LIN {X 0,Y 530.391,Z 772.549,A -85,B 0,C 180,E1 -4220.081,E2 -4220.081} C_VEL
LIN {X 0,Y 530.37,Z 771.261,A -85,B 0,C 180,E1 -4220.851,E2 -4220.851} C_VEL
LIN {X 0,Y 530.472,Z 768.514,A -85,B 0,C 180,E1 -4222.004,E2 -4222.004} C_VEL
LIN {X 0,Y 530.565,Z 764.749,A -85,B 0,C 180,E1 -4223.153,E2 -4223.153} C_VEL
LIN {X 0,Y 530.601,Z 759.88,A -85,B 0,C 180,E1 -4224.299,E2 -4224.299} C_VEL
LIN {X 0,Y 530.713,Z 753.762,A -85,B 0,C 180,E1 -4225.443,E2 -4225.443} C_VEL
LIN {X 0,Y 530.767,Z 746.143,A -85,B 0,C 180,E1 -4226.584,E2 -4226.584} C_VEL
LIN {X 0,Y 531.037,Z 736.67,A -85,B 0,C 180,E1 -4227.725,E2 -4227.725} C_VEL
LIN {X 0,Y 531.27,Z 726.885,A -85,B 0,C 180,E1 -4228.674,E2 -4228.674} C_VEL
LIN {X 0,Y 531.461,Z 715.977,A -85,B 0,C 180,E1 -4229.526,E2 -4229.526} C_VEL
LIN {X 0,Y 531.816,Z 705.381,A -85,B 0,C 180,E1 -4230.189,E2 -4230.189} C_VEL
LIN {X 0,Y 532.07,Z 693.777,A -85,B 0,C 180,E1 -4230.757,E2 -4230.757} C_VEL
LIN {X 0,Y 532.235,Z 680.391,A -85,B 0,C 180,E1 -4231.229,E2 -4231.229} C_VEL
LIN {X 0,Y 532.411,Z 668.005,A -85,B 0,C 180,E1 -4231.513,E2 -4231.513} C_VEL
LIN {X 0,Y 532.675,Z 572.814,A -85,B 0,C 180,E1 -4232.812,E2 -4232.812} C_VEL
LIN {X 0,Y 531.118,Z 564.327,A -85,B 0,C 180,E1 -4232.987,E2 -4232.987} C_VEL
LIN {X 0,Y 531.078,Z 564.336,A -85,B 0,C 180,E1 -4236.077,E2 -4236.077} C_VEL
LIN {X 0,Y 531.019,Z 564.334,A -85,B 0,C 180,E1 -4239.138,E2 -4239.138} C_VEL
LIN {X 0,Y 531.044,Z 564.337,A -85,B 0,C 180,E1 -4242.225,E2 -4242.225} C_VEL
LIN {X 0,Y 530.998,Z 564.337,A -85,B 0,C 180,E1 -4245.349,E2 -4245.349} C_VEL
LIN {X 0,Y 530.991,Z 564.34,A -85,B 0,C 180,E1 -4248.521,E2 -4248.521} C_VEL
LIN {X 0,Y 531.001,Z 564.335,A -85,B 0,C 180,E1 -4250.937,E2 -4250.937} C_VEL
LIN {X 0,Y 530.966,Z 564.347,A -85,B 0,C 180,E1 -4254.225,E2 -4254.225} C_VEL
LIN {X 0,Y 531.006,Z 564.337,A -85,B 0,C 180,E1 -4256.743,E2 -4256.743} C_VEL
LIN {X 0,Y 530.99,Z 564.341,A -85,B 0,C 180,E1 -4259.321,E2 -4259.321} C_VEL
LIN {X 0,Y 531.056,Z 564.335,A -85,B 0,C 180,E1 -4261.1,E2 -4261.1} C_VEL
LIN {X 0,Y 532.797,Z 573.387,A -85,B 0,C 180,E1 -4261.29,E2 -4261.29} C_VEL
LIN {X 0,Y 532.448,Z 668.31,A -85,B 0,C 180,E1 -4262.594,E2 -4262.594} C_VEL
LIN {X 0,Y 532.309,Z 677.915,A -85,B 0,C 180,E1 -4262.8,E2 -4262.8} C_VEL
LIN {X 0,Y 532.099,Z 688.32,A -85,B 0,C 180,E1 -4263.125,E2 -4263.125} C_VEL
LIN {X 0,Y 531.952,Z 697.951,A -85,B 0,C 180,E1 -4263.527,E2 -4263.527} C_VEL
LIN {X 0,Y 531.753,Z 707.979,A -85,B 0,C 180,E1 -4264.059,E2 -4264.059} C_VEL
LIN {X 0,Y 531.543,Z 717.033,A -85,B 0,C 180,E1 -4264.648,E2 -4264.648} C_VEL
LIN {X 0,Y 531.302,Z 725.688,A -85,B 0,C 180,E1 -4265.322,E2 -4265.322} C_VEL
LIN {X 0,Y 531.151,Z 733.257,A -85,B 0,C 180,E1 -4266.019,E2 -4266.019} C_VEL
LIN {X 0,Y 530.967,Z 740.423,A -85,B 0,C 180,E1 -4266.793,E2 -4266.793} C_VEL
LIN {X 0,Y 530.801,Z 747.91,A -85,B 0,C 180,E1 -4267.76,E2 -4267.76} C_VEL
LIN {X 0,Y 530.68,Z 754.502,A -85,B 0,C 180,E1 -4268.788,E2 -4268.788} C_VEL
LIN {X 0,Y 530.604,Z 759.873,A -85,B 0,C 180,E1 -4269.805,E2 -4269.805} C_VEL
LIN {X 0,Y 530.529,Z 762.94,A -85,B 0,C 180,E1 -4270.473,E2 -4270.473} C_VEL
LIN {X 0,Y 530.489,Z 766.691,A -85,B 0,C 180,E1 -4271.482,E2 -4271.482} C_VEL
LIN {X 0,Y 530.427,Z 769.651,A -85,B 0,C 180,E1 -4272.51,E2 -4272.51} C_VEL
LIN {X 0,Y 530.357,Z 771.836,A -85,B 0,C 180,E1 -4273.556,E2 -4273.556} C_VEL
LIN {X 0,Y 530.379,Z 773.243,A -85,B 0,C 180,E1 -4274.61,E2 -4274.61} C_VEL
LIN {X 0,Y 530.38,Z 773.892,A -85,B 0,C 180,E1 -4275.687,E2 -4275.687} C_VEL
LIN {X 0,Y 530.334,Z 773.739,A -85,B 0,C 180,E1 -4276.789,E2 -4276.789} C_VEL
LIN {X 0,Y 530.388,Z 772.739,A -85,B 0,C 180,E1 -4277.904,E2 -4277.904} C_VEL
LIN {X 0,Y 530.375,Z 770.803,A -85,B 0,C 180,E1 -4279.051,E2 -4279.051} C_VEL
LIN {X 0,Y 530.43,Z 767.85,A -85,B 0,C 180,E1 -4280.216,E2 -4280.216} C_VEL
LIN {X 0,Y 530.517,Z 762.445,A -85,B 0,C 180,E1 -4281.733,E2 -4281.733} C_VEL
LIN {X 0,Y 530.587,Z 757.227,A -85,B 0,C 180,E1 -4282.824,E2 -4282.824} C_VEL
LIN {X 0,Y 530.726,Z 751.007,A -85,B 0,C 180,E1 -4283.877,E2 -4283.877} C_VEL
LIN {X 0,Y 530.847,Z 744.546,A -85,B 0,C 180,E1 -4284.79,E2 -4284.79} C_VEL
LIN {X 0,Y 531.056,Z 737.211,A -85,B 0,C 180,E1 -4285.66,E2 -4285.66} C_VEL
LIN {X 0,Y 531.242,Z 728.486,A -85,B 0,C 180,E1 -4286.523,E2 -4286.523} C_VEL
LIN {X 0,Y 531.461,Z 719.636,A -85,B 0,C 180,E1 -4287.252,E2 -4287.252} C_VEL
LIN {X 0,Y 531.674,Z 710.874,A -85,B 0,C 180,E1 -4287.856,E2 -4287.856} C_VEL
LIN {X 0,Y 531.865,Z 701.897,A -85,B 0,C 180,E1 -4288.37,E2 -4288.37} C_VEL
LIN {X 0,Y 532.04,Z 691.985,A -85,B 0,C 180,E1 -4288.825,E2 -4288.825} C_VEL
LIN {X 0,Y 532.229,Z 681.54,A -85,B 0,C 180,E1 -4289.19,E2 -4289.19} C_VEL
LIN {X 0,Y 532.326,Z 671.036,A -85,B 0,C 180,E1 -4289.45,E2 -4289.45} C_VEL
LIN {X 0,Y 532.497,Z 646.041,A -85,B 0,C 180,E1 -4289.817,E2 -4289.817} C_VEL
LIN {X 0,Y 532.659,Z 574.015,A -85,B 0,C 180,E1 -4290.795,E2 -4290.795} C_VEL
LIN {X 0,Y 531.05,Z 565.236,A -85,B 0,C 180,E1 -4290.985,E2 -4290.985} C_VEL
LIN {X 0,Y 530.982,Z 564.345,A -85,B 0,C 180,E1 -4291.244,E2 -4291.244} C_VEL
LIN {X 0,Y 531.008,Z 564.342,A -85,B 0,C 180,E1 -4294.154,E2 -4294.154} C_VEL
LIN {X 0,Y 530.957,Z 564.35,A -85,B 0,C 180,E1 -4296.603,E2 -4296.603} C_VEL
LIN {X 0,Y 531.015,Z 564.337,A -85,B 0,C 180,E1 -4299.872,E2 -4299.872} C_VEL
LIN {X 0,Y 530.983,Z 564.341,A -85,B 0,C 180,E1 -4303.071,E2 -4303.071} C_VEL
LIN {X 0,Y 531.009,Z 564.336,A -85,B 0,C 180,E1 -4305.436,E2 -4305.436} C_VEL
LIN {X 0,Y 531.037,Z 564.34,A -85,B 0,C 180,E1 -4308.55,E2 -4308.55} C_VEL
LIN {X 0,Y 531.052,Z 564.33,A -85,B 0,C 180,E1 -4311.629,E2 -4311.629} C_VEL
LIN {X 0,Y 531.132,Z 564.327,A -85,B 0,C 180,E1 -4314.685,E2 -4314.685} C_VEL
LIN {X 0,Y 531.13,Z 564.32,A -85,B 0,C 180,E1 -4317.725,E2 -4317.725} C_VEL
LIN {X 0,Y 531.146,Z 564.324,A -85,B 0,C 180,E1 -4320.758,E2 -4320.758} C_VEL
LIN {X 0,Y 531.1,Z 564.325,A -85,B 0,C 180,E1 -4323.034,E2 -4323.034} C_VEL
LIN {X 0,Y 531.081,Z 564.329,A -85,B 0,C 180,E1 -4326.077,E2 -4326.077} C_VEL
LIN {X 0,Y 531.027,Z 564.333,A -85,B 0,C 180,E1 -4329.138,E2 -4329.138} C_VEL
LIN {X 0,Y 531.031,Z 564.336,A -85,B 0,C 180,E1 -4332.225,E2 -4332.225} C_VEL
LIN {X 0,Y 530.986,Z 564.337,A -85,B 0,C 180,E1 -4335.35,E2 -4335.35} C_VEL
LIN {X 0,Y 531.007,Z 564.333,A -85,B 0,C 180,E1 -4337.723,E2 -4337.723} C_VEL
LIN {X 0,Y 530.996,Z 564.339,A -85,B 0,C 180,E1 -4340.938,E2 -4340.938} C_VEL
LIN {X 0,Y 530.999,Z 564.338,A -85,B 0,C 180,E1 -4344.046,E2 -4344.046} C_VEL
LIN {X 0,Y 531.004,Z 564.34,A -85,B 0,C 180,E1 -4346.744,E2 -4346.744} C_VEL
LIN {X 0,Y 530.993,Z 564.338,A -85,B 0,C 180,E1 -4349.322,E2 -4349.322} C_VEL
LIN {X 0,Y 530.973,Z 564.343,A -85,B 0,C 180,E1 -4352.104,E2 -4352.104} C_VEL
LIN {X 0,Y 530.984,Z 564.343,A -85,B 0,C 180,E1 -4354.855,E2 -4354.855} C_VEL
LIN {X 0,Y 530.962,Z 564.341,A -85,B 0,C 180,E1 -4357.508,E2 -4357.508} C_VEL
LIN {X 0,Y 531.021,Z 564.342,A -85,B 0,C 180,E1 -4360.429,E2 -4360.429} C_VEL
LIN {X 0,Y 530.963,Z 564.341,A -85,B 0,C 180,E1 -4363.495,E2 -4363.495} C_VEL
LIN {X 0,Y 530.955,Z 564.351,A -85,B 0,C 180,E1 -4366.506,E2 -4366.506} C_VEL
LIN {X 0,Y 530.986,Z 564.341,A -85,B 0,C 180,E1 -4368.977,E2 -4368.977} C_VEL
LIN {X 0,Y 530.957,Z 564.342,A -85,B 0,C 180,E1 -4371.53,E2 -4371.53} C_VEL
LIN {X 0,Y 530.961,Z 564.35,A -85,B 0,C 180,E1 -4374.381,E2 -4374.381} C_VEL
LIN {X 0,Y 530.969,Z 564.343,A -85,B 0,C 180,E1 -4377.134,E2 -4377.134} C_VEL
LIN {X 0,Y 530.968,Z 564.343,A -85,B 0,C 180,E1 -4379.804,E2 -4379.804} C_VEL
LIN {X 0,Y 531.015,Z 564.344,A -85,B 0,C 180,E1 -4382.468,E2 -4382.468} C_VEL
LIN {X 0,Y 531.004,Z 564.377,A -85,B 0,C 180,E1 -4383.519,E2 -4383.519} C_VEL
LIN {X 0,Y 532.974,Z 574.901,A -85,B 0,C 180,E1 -4385.042,E2 -4385.042} C_VEL
LIN {X 0,Y 532.626,Z 593.287,A -85,B 0,C 180,E1 -4387.502,E2 -4387.502} C_VEL
LIN {X 0,Y 532.157,Z 617.709,A -85,B 0,C 180,E1 -4390.722,E2 -4390.722} C_VEL
LIN {X 0,Y 531.683,Z 641.975,A -85,B 0,C 180,E1 -4393.884,E2 -4393.884} C_VEL
LIN {X 0,Y 531.55,Z 650.859,A -85,B 0,C 180,E1 -4395.042,E2 -4395.042} C_VEL
LIN {X 0,Y 532.848,Z 660.029,A -85,B 0,C 180,E1 -4395.204,E2 -4395.204} C_VEL
LIN {X 0,Y 532.474,Z 759.96,A -85,B 0,C 180,E1 -4396.573,E2 -4396.573} C_VEL
LIN {X 0,Y 532.254,Z 772.456,A -85,B 0,C 180,E1 -4396.883,E2 -4396.883} C_VEL
LIN {X 0,Y 532.024,Z 785.368,A -85,B 0,C 180,E1 -4397.362,E2 -4397.362} C_VEL
LIN {X 0,Y 531.807,Z 797.309,A -85,B 0,C 180,E1 -4397.967,E2 -4397.967} C_VEL
LIN {X 0,Y 531.526,Z 809.198,A -85,B 0,C 180,E1 -4398.754,E2 -4398.754} C_VEL
LIN {X 0,Y 531.255,Z 819.607,A -85,B 0,C 180,E1 -4399.616,E2 -4399.616} C_VEL
LIN {X 0,Y 531.06,Z 828.116,A -85,B 0,C 180,E1 -4400.478,E2 -4400.478} C_VEL
LIN {X 0,Y 530.886,Z 835.962,A -85,B 0,C 180,E1 -4401.435,E2 -4401.435} C_VEL
LIN {X 0,Y 530.685,Z 843.623,A -85,B 0,C 180,E1 -4402.581,E2 -4402.581} C_VEL
LIN {X 0,Y 530.604,Z 850.679,A -85,B 0,C 180,E1 -4403.918,E2 -4403.918} C_VEL
LIN {X 0,Y 530.459,Z 855.372,A -85,B 0,C 180,E1 -4405.06,E2 -4405.06} C_VEL
LIN {X 0,Y 530.516,Z 858.961,A -85,B 0,C 180,E1 -4406.202,E2 -4406.202} C_VEL
LIN {X 0,Y 530.457,Z 860.81,A -85,B 0,C 180,E1 -4406.962,E2 -4406.962} C_VEL
LIN {X 0,Y 530.41,Z 862.197,A -85,B 0,C 180,E1 -4407.722,E2 -4407.722} C_VEL
LIN {X 0,Y 530.344,Z 863.786,A -85,B 0,C 180,E1 -4409.241,E2 -4409.241} C_VEL
LIN {X 0,Y 530.342,Z 864,A -85,B 0,C 180,E1 -4410,E2 -4410} C_VEL
LIN {X 0,Y 530.361,Z 863.183,A -85,B 0,C 180,E1 -4411.519,E2 -4411.519} C_VEL
LIN {X 0,Y 530.41,Z 862.194,A -85,B 0,C 180,E1 -4412.278,E2 -4412.278} C_VEL
LIN {X 0,Y 530.457,Z 860.807,A -85,B 0,C 180,E1 -4413.038,E2 -4413.038} C_VEL
LIN {X 0,Y 530.523,Z 857.895,A -85,B 0,C 180,E1 -4414.178,E2 -4414.178} C_VEL
LIN {X 0,Y 530.525,Z 853.95,A -85,B 0,C 180,E1 -4415.321,E2 -4415.321} C_VEL
LIN {X 0,Y 530.599,Z 848.264,A -85,B 0,C 180,E1 -4416.582,E2 -4416.582} C_VEL
LIN {X 0,Y 530.758,Z 841.237,A -85,B 0,C 180,E1 -4417.8,E2 -4417.8} C_VEL
LIN {X 0,Y 530.93,Z 832.994,A -85,B 0,C 180,E1 -4418.948,E2 -4418.948} C_VEL
LIN {X 0,Y 531.137,Z 824.542,A -85,B 0,C 180,E1 -4419.905,E2 -4419.905} C_VEL
LIN {X 0,Y 531.408,Z 814.096,A -85,B 0,C 180,E1 -4420.863,E2 -4420.863} C_VEL
LIN {X 0,Y 531.667,Z 802.16,A -85,B 0,C 180,E1 -4421.737,E2 -4421.737} C_VEL
LIN {X 0,Y 531.95,Z 790.496,A -85,B 0,C 180,E1 -4422.397,E2 -4422.397} C_VEL
LIN {X 0,Y 532.205,Z 778.182,A -85,B 0,C 180,E1 -4422.924,E2 -4422.924} C_VEL
LIN {X 0,Y 532.353,Z 765.533,A -85,B 0,C 180,E1 -4423.309,E2 -4423.309} C_VEL
LIN {X 0,Y 532.491,Z 752.335,A -85,B 0,C 180,E1 -4423.548,E2 -4423.548} C_VEL
LIN {X 0,Y 532.701,Z 656.891,A -85,B 0,C 180,E1 -4424.843,E2 -4424.843} C_VEL
LIN {X 0,Y 531.719,Z 649.794,A -85,B 0,C 180,E1 -4424.977,E2 -4424.977} C_VEL
LIN {X 0,Y 532.246,Z 621.608,A -85,B 0,C 180,E1 -4428.199,E2 -4428.199} C_VEL
LIN {X 0,Y 532.815,Z 595.021,A -85,B 0,C 180,E1 -4431.268,E2 -4431.268} C_VEL
LIN {X 0,Y 533.193,Z 575.94,A -85,B 0,C 180,E1 -4433.498,E2 -4433.498} C_VEL
LIN {X 0,Y 532.837,Z 572.446,A -85,B 0,C 180,E1 -4433.927,E2 -4433.927} C_VEL
LIN {X 0,Y 531.05,Z 564.336,A -85,B 0,C 180,E1 -4435.002,E2 -4435.002} C_VEL
LIN {X 0,Y 531.018,Z 564.34,A -85,B 0,C 180,E1 -4437.595,E2 -4437.595} C_VEL
LIN {X 0,Y 530.973,Z 564.341,A -85,B 0,C 180,E1 -4440.644,E2 -4440.644} C_VEL
LIN {X 0,Y 530.992,Z 564.344,A -85,B 0,C 180,E1 -4443.771,E2 -4443.771} C_VEL
LIN {X 0,Y 530.966,Z 564.343,A -85,B 0,C 180,E1 -4446.557,E2 -4446.557} C_VEL
LIN {X 0,Y 531.004,Z 564.341,A -85,B 0,C 180,E1 -4449.857,E2 -4449.857} C_VEL
LIN {X 0,Y 530.977,Z 564.343,A -85,B 0,C 180,E1 -4452.456,E2 -4452.456} C_VEL
LIN {X 0,Y 530.983,Z 564.339,A -85,B 0,C 180,E1 -4455.62,E2 -4455.62} C_VEL
LIN {X 0,Y 531.004,Z 564.338,A -85,B 0,C 180,E1 -4458.565,E2 -4458.565} C_VEL
LIN {X 0,Y 530.964,Z 564.339,A -85,B 0,C 180,E1 -4461.345,E2 -4461.345} C_VEL
LIN {X 0,Y 530.976,Z 564.343,A -85,B 0,C 180,E1 -4464.381,E2 -4464.381} C_VEL
LIN {X 0,Y 530.965,Z 564.34,A -85,B 0,C 180,E1 -4467.133,E2 -4467.133} C_VEL
LIN {X 0,Y 530.978,Z 564.34,A -85,B 0,C 180,E1 -4469.803,E2 -4469.803} C_VEL
LIN {X 0,Y 531.01,Z 564.343,A -85,B 0,C 180,E1 -4472.466,E2 -4472.466} C_VEL
LIN {X 0,Y 530.999,Z 564.337,A -85,B 0,C 180,E1 -4474.942,E2 -4474.942} C_VEL
LIN {X 0,Y 530.962,Z 564.342,A -85,B 0,C 180,E1 -4478.246,E2 -4478.246} C_VEL
LIN {X 0,Y 530.988,Z 564.343,A -85,B 0,C 180,E1 -4480.677,E2 -4480.677} C_VEL
LIN {X 0,Y 530.982,Z 564.336,A -85,B 0,C 180,E1 -4483.071,E2 -4483.071} C_VEL
LIN {X 0,Y 531.009,Z 564.333,A -85,B 0,C 180,E1 -4485.436,E2 -4485.436} C_VEL
LIN {X 0,Y 531.037,Z 564.34,A -85,B 0,C 180,E1 -4488.55,E2 -4488.55} C_VEL
LIN {X 0,Y 531.05,Z 564.325,A -85,B 0,C 180,E1 -4491.629,E2 -4491.629} C_VEL
LIN {X 0,Y 531.136,Z 564.328,A -85,B 0,C 180,E1 -4494.685,E2 -4494.685} C_VEL
LIN {X 0,Y 531.13,Z 564.315,A -85,B 0,C 180,E1 -4497.725,E2 -4497.725} C_VEL
LIN {X 0,Y 531.148,Z 564.326,A -85,B 0,C 180,E1 -4500.758,E2 -4500.758} C_VEL
LIN {X 0,Y 531.1,Z 564.327,A -85,B 0,C 180,E1 -4503.034,E2 -4503.034} C_VEL
LIN {X 0,Y 531.081,Z 564.321,A -85,B 0,C 180,E1 -4506.077,E2 -4506.077} C_VEL
LIN {X 0,Y 531.027,Z 564.337,A -85,B 0,C 180,E1 -4509.138,E2 -4509.138} C_VEL
LIN {X 0,Y 531.031,Z 564.33,A -85,B 0,C 180,E1 -4512.225,E2 -4512.225} C_VEL
LIN {X 0,Y 530.986,Z 564.341,A -85,B 0,C 180,E1 -4515.35,E2 -4515.35} C_VEL
LIN {X 0,Y 531.007,Z 564.333,A -85,B 0,C 180,E1 -4517.723,E2 -4517.723} C_VEL
LIN {X 0,Y 530.993,Z 564.344,A -85,B 0,C 180,E1 -4520.938,E2 -4520.938} C_VEL
LIN {X 0,Y 530.971,Z 564.337,A -85,B 0,C 180,E1 -4524.225,E2 -4524.225} C_VEL
LIN {X 0,Y 531.004,Z 564.339,A -85,B 0,C 180,E1 -4526.744,E2 -4526.744} C_VEL
LIN {X 0,Y 530.992,Z 564.34,A -85,B 0,C 180,E1 -4529.322,E2 -4529.322} C_VEL
LIN {X 0,Y 530.972,Z 564.34,A -85,B 0,C 180,E1 -4532.104,E2 -4532.104} C_VEL
LIN {X 0,Y 530.981,Z 564.341,A -85,B 0,C 180,E1 -4534.855,E2 -4534.855} C_VEL
LIN {X 0,Y 530.967,Z 564.345,A -85,B 0,C 180,E1 -4537.508,E2 -4537.508} C_VEL
LIN {X 0,Y 530.979,Z 564.338,A -85,B 0,C 180,E1 -4540.433,E2 -4540.433} C_VEL
LIN {X 0,Y 530.966,Z 564.343,A -85,B 0,C 180,E1 -4543.283,E2 -4543.283} C_VEL
LIN {X 0,Y 530.959,Z 564.346,A -85,B 0,C 180,E1 -4543.581,E2 -4543.581} C_VEL
LIN {X 0,Y 530.285,Z 564.427,A -85,B 0,C 180,E1 -4544.214,E2 -4544.214} C_VEL
LIN {X 0,Y 527.432,Z 564.789,A -85,B 0,C 180,E1 -4545.243,E2 -4545.243} C_VEL
LIN {X 0,Y 525.026,Z 565.087,A -85,B 0,C 180,E1 -4546.071,E2 -4546.071} C_VEL
LIN {X 0,Y 523.994,Z 565.211,A -85,B 0,C 180,E1 -4546.711,E2 -4546.711} C_VEL
LIN {X 0,Y 523.91,Z 565.22,A -85,B 0,C 180,E1 -4546.928,E2 -4546.928} C_VEL
LIN {X 0,Y 523.945,Z 565.218,A -85,B 0,C 180,E1 -4549.921,E2 -4549.921} C_VEL
LIN {X 0,Y 523.909,Z 565.219,A -85,B 0,C 180,E1 -4552.869,E2 -4552.869} C_VEL
LIN {X 0,Y 523.942,Z 565.221,A -85,B 0,C 180,E1 -4555.711,E2 -4555.711} C_VEL
LIN {X 0,Y 523.922,Z 565.218,A -85,B 0,C 180,E1 -4558.457,E2 -4558.457} C_VEL
LIN {X 0,Y 523.939,Z 565.221,A -85,B 0,C 180,E1 -4561.126,E2 -4561.126} C_VEL
LIN {X 0,Y 523.961,Z 565.371,A -85,B 0,C 180,E1 -4562.868,E2 -4562.868} C_VEL
LIN {X 0,Y 523.989,Z 565.59,A -85,B 0,C 180,E1 -4562.918,E2 -4562.918} C_VEL
LIN {X 0,Y 525.93,Z 575.467,A -85,B 0,C 180,E1 -4563.114,E2 -4563.114} C_VEL
LIN {X 0,Y 525.487,Z 671.22,A -85,B 0,C 180,E1 -4564.449,E2 -4564.449} C_VEL
LIN {X 0,Y 525.28,Z 683.407,A -85,B 0,C 180,E1 -4564.757,E2 -4564.757} C_VEL
LIN {X 0,Y 525.143,Z 695.77,A -85,B 0,C 180,E1 -4565.226,E2 -4565.226} C_VEL
LIN {X 0,Y 524.907,Z 707.21,A -85,B 0,C 180,E1 -4565.812,E2 -4565.812} C_VEL
LIN {X 0,Y 524.603,Z 717.948,A -85,B 0,C 180,E1 -4566.513,E2 -4566.513} C_VEL
LIN {X 0,Y 524.309,Z 727.575,A -85,B 0,C 180,E1 -4567.291,E2 -4567.291} C_VEL
LIN {X 0,Y 524.093,Z 736.326,A -85,B 0,C 180,E1 -4568.154,E2 -4568.154} C_VEL
LIN {X 0,Y 523.853,Z 744.814,A -85,B 0,C 180,E1 -4569.175,E2 -4569.175} C_VEL
LIN {X 0,Y 523.661,Z 753.01,A -85,B 0,C 180,E1 -4570.396,E2 -4570.396} C_VEL
LIN {X 0,Y 523.533,Z 759.515,A -85,B 0,C 180,E1 -4571.611,E2 -4571.611} C_VEL
LIN {X 0,Y 523.445,Z 764.578,A -85,B 0,C 180,E1 -4572.82,E2 -4572.82} C_VEL
LIN {X 0,Y 523.355,Z 768.482,A -85,B 0,C 180,E1 -4574.021,E2 -4574.021} C_VEL
LIN {X 0,Y 523.339,Z 771.289,A -85,B 0,C 180,E1 -4575.218,E2 -4575.218} C_VEL
LIN {X 0,Y 523.3,Z 772.591,A -85,B 0,C 180,E1 -4576.011,E2 -4576.011} C_VEL
LIN {X 0,Y 523.268,Z 773.482,A -85,B 0,C 180,E1 -4576.802,E2 -4576.802} C_VEL
LIN {X 0,Y 523.282,Z 773.913,A -85,B 0,C 180,E1 -4577.591,E2 -4577.591} C_VEL
LIN {X 0,Y 523.363,Z 773.892,A -85,B 0,C 180,E1 -4578.604,E2 -4578.604} C_VEL
LIN {X 0,Y 523.31,Z 772.783,A -85,B 0,C 180,E1 -4579.946,E2 -4579.946} C_VEL
LIN {X 0,Y 523.316,Z 769.939,A -85,B 0,C 180,E1 -4581.505,E2 -4581.505} C_VEL
LIN {X 0,Y 523.451,Z 766.663,A -85,B 0,C 180,E1 -4582.672,E2 -4582.672} C_VEL
LIN {X 0,Y 523.434,Z 762.367,A -85,B 0,C 180,E1 -4583.834,E2 -4583.834} C_VEL
LIN {X 0,Y 523.543,Z 755.905,A -85,B 0,C 180,E1 -4585.187,E2 -4585.187} C_VEL
LIN {X 0,Y 523.722,Z 748.867,A -85,B 0,C 180,E1 -4586.345,E2 -4586.345} C_VEL
LIN {X 0,Y 523.954,Z 740.148,A -85,B 0,C 180,E1 -4587.502,E2 -4587.502} C_VEL
LIN {X 0,Y 524.225,Z 730.125,A -85,B 0,C 180,E1 -4588.56,E2 -4588.56} C_VEL
LIN {X 0,Y 524.451,Z 720.028,A -85,B 0,C 180,E1 -4589.424,E2 -4589.424} C_VEL
LIN {X 0,Y 524.8,Z 708.697,A -85,B 0,C 180,E1 -4590.192,E2 -4590.192} C_VEL
LIN {X 0,Y 525.165,Z 695.762,A -85,B 0,C 180,E1 -4590.863,E2 -4590.863} C_VEL
LIN {X 0,Y 525.351,Z 683.831,A -85,B 0,C 180,E1 -4591.317,E2 -4591.317} C_VEL
LIN {X 0,Y 525.548,Z 670.515,A -85,B 0,C 180,E1 -4591.652,E2 -4591.652} C_VEL
LIN {X 0,Y 525.827,Z 573.57,A -85,B 0,C 180,E1 -4593.005,E2 -4593.005} C_VEL
LIN {X 0,Y 524.47,Z 566.934,A -85,B 0,C 180,E1 -4593.138,E2 -4593.138} C_VEL
LIN {X 0,Y 524.03,Z 565.211,A -85,B 0,C 180,E1 -4593.195,E2 -4593.195} C_VEL
LIN {X 0,Y 524.04,Z 565.212,A -85,B 0,C 180,E1 -4596.159,E2 -4596.159} C_VEL
LIN {X 0,Y 523.989,Z 565.211,A -85,B 0,C 180,E1 -4599.262,E2 -4599.262} C_VEL
LIN {X 0,Y 524.028,Z 565.209,A -85,B 0,C 180,E1 -4601.751,E2 -4601.751} C_VEL
LIN {X 0,Y 523.996,Z 565.209,A -85,B 0,C 180,E1 -4605.052,E2 -4605.052} C_VEL
LIN {X 0,Y 523.966,Z 565.221,A -85,B 0,C 180,E1 -4607.968,E2 -4607.968} C_VEL
LIN {X 0,Y 523.974,Z 565.215,A -85,B 0,C 180,E1 -4610.409,E2 -4610.409} C_VEL
LIN {X 0,Y 523.912,Z 565.219,A -85,B 0,C 180,E1 -4612.893,E2 -4612.893} C_VEL
LIN {X 0,Y 523.985,Z 565.219,A -85,B 0,C 180,E1 -4616.019,E2 -4616.019} C_VEL
LIN {X 0,Y 523.942,Z 565.218,A -85,B 0,C 180,E1 -4618.874,E2 -4618.874} C_VEL
LIN {X 0,Y 524.023,Z 565.211,A -85,B 0,C 180,E1 -4620.911,E2 -4620.911} C_VEL
LIN {X 0,Y 525.834,Z 573.683,A -85,B 0,C 180,E1 -4621.09,E2 -4621.09} C_VEL
LIN {X 0,Y 525.495,Z 670.324,A -85,B 0,C 180,E1 -4622.443,E2 -4622.443} C_VEL
LIN {X 0,Y 525.388,Z 680.701,A -85,B 0,C 180,E1 -4622.69,E2 -4622.69} C_VEL
LIN {X 0,Y 525.224,Z 690.839,A -85,B 0,C 180,E1 -4623.034,E2 -4623.034} C_VEL
LIN {X 0,Y 524.988,Z 701.004,A -85,B 0,C 180,E1 -4623.487,E2 -4623.487} C_VEL
LIN {X 0,Y 524.796,Z 710.378,A -85,B 0,C 180,E1 -4624.015,E2 -4624.015} C_VEL
LIN {X 0,Y 524.566,Z 718.82,A -85,B 0,C 180,E1 -4624.591,E2 -4624.591} C_VEL
LIN {X 0,Y 524.342,Z 726.302,A -85,B 0,C 180,E1 -4625.193,E2 -4625.193} C_VEL
LIN {X 0,Y 524.149,Z 733.941,A -85,B 0,C 180,E1 -4625.916,E2 -4625.916} C_VEL
LIN {X 0,Y 523.95,Z 741.311,A -85,B 0,C 180,E1 -4626.741,E2 -4626.741} C_VEL
LIN {X 0,Y 523.755,Z 748.192,A -85,B 0,C 180,E1 -4627.656,E2 -4627.656} C_VEL
LIN {X 0,Y 523.622,Z 754.623,A -85,B 0,C 180,E1 -4628.687,E2 -4628.687} C_VEL
LIN {X 0,Y 523.545,Z 759.332,A -85,B 0,C 180,E1 -4629.588,E2 -4629.588} C_VEL
LIN {X 0,Y 523.436,Z 763.807,A -85,B 0,C 180,E1 -4630.63,E2 -4630.63} C_VEL
LIN {X 0,Y 523.389,Z 767.452,A -85,B 0,C 180,E1 -4631.678,E2 -4631.678} C_VEL
LIN {X 0,Y 523.333,Z 769.437,A -85,B 0,C 180,E1 -4632.386,E2 -4632.386} C_VEL
LIN {X 0,Y 523.258,Z 771.8,A -85,B 0,C 180,E1 -4633.507,E2 -4633.507} C_VEL
LIN {X 0,Y 523.279,Z 773.266,A -85,B 0,C 180,E1 -4634.616,E2 -4634.616} C_VEL
LIN {X 0,Y 523.279,Z 773.892,A -85,B 0,C 180,E1 -4635.701,E2 -4635.701} C_VEL
LIN {X 0,Y 523.239,Z 773.746,A -85,B 0,C 180,E1 -4636.763,E2 -4636.763} C_VEL
LIN {X 0,Y 523.309,Z 772.863,A -85,B 0,C 180,E1 -4637.817,E2 -4637.817} C_VEL
LIN {X 0,Y 523.305,Z 770.274,A -85,B 0,C 180,E1 -4639.356,E2 -4639.356} C_VEL
LIN {X 0,Y 523.402,Z 765.974,A -85,B 0,C 180,E1 -4640.869,E2 -4640.869} C_VEL
LIN {X 0,Y 523.471,Z 760.957,A -85,B 0,C 180,E1 -4642.146,E2 -4642.146} C_VEL
LIN {X 0,Y 523.553,Z 756.582,A -85,B 0,C 180,E1 -4643.052,E2 -4643.052} C_VEL
LIN {X 0,Y 523.706,Z 750.78,A -85,B 0,C 180,E1 -4644.047,E2 -4644.047} C_VEL
LIN {X 0,Y 523.874,Z 743.466,A -85,B 0,C 180,E1 -4645.081,E2 -4645.081} C_VEL
LIN {X 0,Y 524.104,Z 736.851,A -85,B 0,C 180,E1 -4645.867,E2 -4645.867} C_VEL
LIN {X 0,Y 524.292,Z 728.984,A -85,B 0,C 180,E1 -4646.661,E2 -4646.661} C_VEL
LIN {X 0,Y 524.525,Z 720.38,A -85,B 0,C 180,E1 -4647.387,E2 -4647.387} C_VEL
LIN {X 0,Y 524.766,Z 710.679,A -85,B 0,C 180,E1 -4648.061,E2 -4648.061} C_VEL
LIN {X 0,Y 524.967,Z 701.452,A -85,B 0,C 180,E1 -4648.585,E2 -4648.585} C_VEL
LIN {X 0,Y 525.158,Z 691.073,A -85,B 0,C 180,E1 -4649.052,E2 -4649.052} C_VEL
LIN {X 0,Y 525.334,Z 680.742,A -85,B 0,C 180,E1 -4649.402,E2 -4649.402} C_VEL
LIN {X 0,Y 525.471,Z 670.156,A -85,B 0,C 180,E1 -4649.652,E2 -4649.652} C_VEL
LIN {X 0,Y 525.874,Z 575.325,A -85,B 0,C 180,E1 -4650.976,E2 -4650.976} C_VEL
LIN {X 0,Y 524.083,Z 566.116,A -85,B 0,C 180,E1 -4651.161,E2 -4651.161} C_VEL
LIN {X 0,Y 523.96,Z 565.22,A -85,B 0,C 180,E1 -4651.4,E2 -4651.4} C_VEL
LIN {X 0,Y 523.977,Z 565.216,A -85,B 0,C 180,E1 -4653.979,E2 -4653.979} C_VEL
LIN {X 0,Y 523.928,Z 565.224,A -85,B 0,C 180,E1 -4656.27,E2 -4656.27} C_VEL
LIN {X 0,Y 523.938,Z 565.223,A -85,B 0,C 180,E1 -4658.766,E2 -4658.766} C_VEL
LIN {X 0,Y 523.945,Z 565.217,A -85,B 0,C 180,E1 -4661.22,E2 -4661.22} C_VEL
LIN {X 0,Y 523.931,Z 565.218,A -85,B 0,C 180,E1 -4663.639,E2 -4663.639} C_VEL
LIN {X 0,Y 523.932,Z 565.22,A -85,B 0,C 180,E1 -4666.028,E2 -4666.028} C_VEL
LIN {X 0,Y 524.001,Z 565.216,A -85,B 0,C 180,E1 -4668.394,E2 -4668.394} C_VEL
LIN {X 0,Y 523.999,Z 565.209,A -85,B 0,C 180,E1 -4671.516,E2 -4671.516} C_VEL
LIN {X 0,Y 524.09,Z 565.204,A -85,B 0,C 180,E1 -4674.614,E2 -4674.614} C_VEL
LIN {X 0,Y 524.102,Z 565.195,A -85,B 0,C 180,E1 -4677.694,E2 -4677.694} C_VEL
LIN {X 0,Y 524.115,Z 565.2,A -85,B 0,C 180,E1 -4680.768,E2 -4680.768} C_VEL
LIN {X 0,Y 524.067,Z 565.2,A -85,B 0,C 180,E1 -4683.075,E2 -4683.075} C_VEL
LIN {X 0,Y 524.042,Z 565.207,A -85,B 0,C 180,E1 -4686.159,E2 -4686.159} C_VEL
LIN {X 0,Y 523.995,Z 565.208,A -85,B 0,C 180,E1 -4689.262,E2 -4689.262} C_VEL
LIN {X 0,Y 524.014,Z 565.206,A -85,B 0,C 180,E1 -4691.752,E2 -4691.752} C_VEL
LIN {X 0,Y 523.983,Z 565.211,A -85,B 0,C 180,E1 -4695.053,E2 -4695.053} C_VEL
LIN {X 0,Y 523.955,Z 565.213,A -85,B 0,C 180,E1 -4697.969,E2 -4697.969} C_VEL
LIN {X 0,Y 523.964,Z 565.218,A -85,B 0,C 180,E1 -4700.41,E2 -4700.41} C_VEL
LIN {X 0,Y 523.935,Z 565.218,A -85,B 0,C 180,E1 -4702.893,E2 -4702.893} C_VEL
LIN {X 0,Y 523.977,Z 565.214,A -85,B 0,C 180,E1 -4706.021,E2 -4706.021} C_VEL
LIN {X 0,Y 523.944,Z 565.219,A -85,B 0,C 180,E1 -4708.875,E2 -4708.875} C_VEL
LIN {X 0,Y 523.925,Z 565.217,A -85,B 0,C 180,E1 -4711.544,E2 -4711.544} C_VEL
LIN {X 0,Y 523.939,Z 565.221,A -85,B 0,C 180,E1 -4714.29,E2 -4714.29} C_VEL
LIN {X 0,Y 523.907,Z 565.221,A -85,B 0,C 180,E1 -4717.132,E2 -4717.132} C_VEL
LIN {X 0,Y 523.963,Z 565.216,A -85,B 0,C 180,E1 -4720.135,E2 -4720.135} C_VEL
LIN {X 0,Y 523.921,Z 565.219,A -85,B 0,C 180,E1 -4723.167,E2 -4723.167} C_VEL
LIN {X 0,Y 523.934,Z 565.218,A -85,B 0,C 180,E1 -4725.773,E2 -4725.773} C_VEL
LIN {X 0,Y 523.941,Z 565.219,A -85,B 0,C 180,E1 -4728.909,E2 -4728.909} C_VEL
LIN {X 0,Y 523.914,Z 565.222,A -85,B 0,C 180,E1 -4731.899,E2 -4731.899} C_VEL
LIN {X 0,Y 523.931,Z 565.221,A -85,B 0,C 180,E1 -4734.911,E2 -4734.911} C_VEL
LIN {X 0,Y 523.936,Z 565.218,A -85,B 0,C 180,E1 -4737.68,E2 -4737.68} C_VEL
LIN {X 0,Y 523.953,Z 565.222,A -85,B 0,C 180,E1 -4740.677,E2 -4740.677} C_VEL
LIN {X 0,Y 523.983,Z 565.293,A -85,B 0,C 180,E1 -4743.354,E2 -4743.354} C_VEL
LIN {X 0,Y 526.011,Z 575.584,A -85,B 0,C 180,E1 -4744.87,E2 -4744.87} C_VEL
LIN {X 0,Y 525.663,Z 594.229,A -85,B 0,C 180,E1 -4747.405,E2 -4747.405} C_VEL
LIN {X 0,Y 525.143,Z 618.575,A -85,B 0,C 180,E1 -4750.657,E2 -4750.657} C_VEL
LIN {X 0,Y 524.606,Z 644.352,A -85,B 0,C 180,E1 -4754.06,E2 -4754.06} C_VEL
LIN {X 0,Y 524.552,Z 650.359,A -85,B 0,C 180,E1 -4754.842,E2 -4754.842} C_VEL
LIN {X 0,Y 525.974,Z 660.389,A -85,B 0,C 180,E1 -4755.02,E2 -4755.02} C_VEL
LIN {X 0,Y 525.566,Z 759.614,A -85,B 0,C 180,E1 -4756.393,E2 -4756.393} C_VEL
LIN {X 0,Y 525.341,Z 772.21,A -85,B 0,C 180,E1 -4756.707,E2 -4756.707} C_VEL
LIN {X 0,Y 525.106,Z 785.234,A -85,B 0,C 180,E1 -4757.193,E2 -4757.193} C_VEL
LIN {X 0,Y 524.828,Z 797.797,A -85,B 0,C 180,E1 -4757.836,E2 -4757.836} C_VEL
LIN {X 0,Y 524.554,Z 809.197,A -85,B 0,C 180,E1 -4758.602,E2 -4758.602} C_VEL
LIN {X 0,Y 524.241,Z 819.606,A -85,B 0,C 180,E1 -4759.476,E2 -4759.476} C_VEL
LIN {X 0,Y 524.054,Z 828.116,A -85,B 0,C 180,E1 -4760.35,E2 -4760.35} C_VEL
LIN {X 0,Y 523.852,Z 835.962,A -85,B 0,C 180,E1 -4761.319,E2 -4761.319} C_VEL
LIN {X 0,Y 523.633,Z 843.623,A -85,B 0,C 180,E1 -4762.481,E2 -4762.481} C_VEL
LIN {X 0,Y 523.515,Z 850.679,A -85,B 0,C 180,E1 -4763.835,E2 -4763.835} C_VEL
LIN {X 0,Y 523.384,Z 855.372,A -85,B 0,C 180,E1 -4764.993,E2 -4764.993} C_VEL
LIN {X 0,Y 523.443,Z 858.961,A -85,B 0,C 180,E1 -4766.151,E2 -4766.151} C_VEL
LIN {X 0,Y 523.368,Z 860.81,A -85,B 0,C 180,E1 -4766.921,E2 -4766.921} C_VEL
LIN {X 0,Y 523.334,Z 862.196,A -85,B 0,C 180,E1 -4767.691,E2 -4767.691} C_VEL
LIN {X 0,Y 523.25,Z 863.786,A -85,B 0,C 180,E1 -4769.23,E2 -4769.23} C_VEL
LIN {X 0,Y 523.246,Z 864,A -85,B 0,C 180,E1 -4770,E2 -4770} C_VEL
LIN {X 0,Y 523.274,Z 863.182,A -85,B 0,C 180,E1 -4771.539,E2 -4771.539} C_VEL
LIN {X 0,Y 523.334,Z 862.193,A -85,B 0,C 180,E1 -4772.309,E2 -4772.309} C_VEL
LIN {X 0,Y 523.368,Z 860.807,A -85,B 0,C 180,E1 -4773.079,E2 -4773.079} C_VEL
LIN {X 0,Y 523.442,Z 857.894,A -85,B 0,C 180,E1 -4774.235,E2 -4774.235} C_VEL
LIN {X 0,Y 523.464,Z 853.95,A -85,B 0,C 180,E1 -4775.393,E2 -4775.393} C_VEL
LIN {X 0,Y 523.523,Z 848.728,A -85,B 0,C 180,E1 -4776.581,E2 -4776.581} C_VEL
LIN {X 0,Y 523.665,Z 842.467,A -85,B 0,C 180,E1 -4777.713,E2 -4777.713} C_VEL
LIN {X 0,Y 523.856,Z 834.479,A -85,B 0,C 180,E1 -4778.875,E2 -4778.875} C_VEL
LIN {X 0,Y 524.107,Z 826.335,A -85,B 0,C 180,E1 -4779.844,E2 -4779.844} C_VEL
LIN {X 0,Y 524.366,Z 816.4,A -85,B 0,C 180,E1 -4780.815,E2 -4780.815} C_VEL
LIN {X 0,Y 524.663,Z 805.192,A -85,B 0,C 180,E1 -4781.688,E2 -4781.688} C_VEL
LIN {X 0,Y 524.921,Z 794.132,A -85,B 0,C 180,E1 -4782.369,E2 -4782.369} C_VEL
LIN {X 0,Y 525.206,Z 781.845,A -85,B 0,C 180,E1 -4782.952,E2 -4782.952} C_VEL
LIN {X 0,Y 525.372,Z 768.939,A -85,B 0,C 180,E1 -4783.39,E2 -4783.39} C_VEL
LIN {X 0,Y 525.595,Z 755.265,A -85,B 0,C 180,E1 -4783.68,E2 -4783.68} C_VEL
LIN {X 0,Y 525.945,Z 658.838,A -85,B 0,C 180,E1 -4785.003,E2 -4785.003} C_VEL
LIN {X 0,Y 524.716,Z 649.354,A -85,B 0,C 180,E1 -4785.177,E2 -4785.177} C_VEL
LIN {X 0,Y 525.267,Z 621.564,A -85,B 0,C 180,E1 -4788.394,E2 -4788.394} C_VEL
LIN {X 0,Y 525.878,Z 596.227,A -85,B 0,C 180,E1 -4791.356,E2 -4791.356} C_VEL
LIN {X 0,Y 526.305,Z 577.154,A -85,B 0,C 180,E1 -4793.615,E2 -4793.615} C_VEL
LIN {X 0,Y 525.594,Z 572.667,A -85,B 0,C 180,E1 -4794.189,E2 -4794.189} C_VEL
LIN {X 0,Y 524.001,Z 565.215,A -85,B 0,C 180,E1 -4795.203,E2 -4795.203} C_VEL
LIN {X 0,Y 523.971,Z 565.22,A -85,B 0,C 180,E1 -4797.998,E2 -4797.998} C_VEL
LIN {X 0,Y 523.944,Z 565.216,A -85,B 0,C 180,E1 -4800.854,E2 -4800.854} C_VEL
LIN {X 0,Y 523.962,Z 565.219,A -85,B 0,C 180,E1 -4803.734,E2 -4803.734} C_VEL
LIN {X 0,Y 523.921,Z 565.222,A -85,B 0,C 180,E1 -4806.404,E2 -4806.404} C_VEL
LIN {X 0,Y 523.929,Z 565.216,A -85,B 0,C 180,E1 -4809.083,E2 -4809.083} C_VEL
LIN {X 0,Y 523.969,Z 565.212,A -85,B 0,C 180,E1 -4811.312,E2 -4811.312} C_VEL
LIN {X 0,Y 523.952,Z 565.215,A -85,B 0,C 180,E1 -4814.691,E2 -4814.691} C_VEL
LIN {X 0,Y 523.954,Z 565.219,A -85,B 0,C 180,E1 -4817.881,E2 -4817.881} C_VEL
LIN {X 0,Y 523.955,Z 565.213,A -85,B 0,C 180,E1 -4820.918,E2 -4820.918} C_VEL
LIN {X 0,Y 523.923,Z 565.221,A -85,B 0,C 180,E1 -4823.827,E2 -4823.827} C_VEL
LIN {X 0,Y 523.935,Z 565.22,A -85,B 0,C 180,E1 -4826.635,E2 -4826.635} C_VEL
LIN {X 0,Y 523.956,Z 565.213,A -85,B 0,C 180,E1 -4829.356,E2 -4829.356} C_VEL
LIN {X 0,Y 523.972,Z 565.216,A -85,B 0,C 180,E1 -4832.28,E2 -4832.28} C_VEL
LIN {X 0,Y 523.947,Z 565.22,A -85,B 0,C 180,E1 -4834.581,E2 -4834.581} C_VEL
LIN {X 0,Y 523.907,Z 565.215,A -85,B 0,C 180,E1 -4837.106,E2 -4837.106} C_VEL
LIN {X 0,Y 523.97,Z 565.213,A -85,B 0,C 180,E1 -4839.865,E2 -4839.865} C_VEL
LIN {X 0,Y 523.961,Z 565.213,A -85,B 0,C 180,E1 -4842.837,E2 -4842.837} C_VEL
LIN {X 0,Y 523.966,Z 565.211,A -85,B 0,C 180,E1 -4845.235,E2 -4845.235} C_VEL
LIN {X 0,Y 524.001,Z 565.215,A -85,B 0,C 180,E1 -4848.394,E2 -4848.394} C_VEL
LIN {X 0,Y 523.998,Z 565.203,A -85,B 0,C 180,E1 -4851.516,E2 -4851.516} C_VEL
LIN {X 0,Y 524.094,Z 565.205,A -85,B 0,C 180,E1 -4854.614,E2 -4854.614} C_VEL
LIN {X 0,Y 524.102,Z 565.191,A -85,B 0,C 180,E1 -4857.694,E2 -4857.694} C_VEL
LIN {X 0,Y 524.117,Z 565.201,A -85,B 0,C 180,E1 -4860.768,E2 -4860.768} C_VEL
LIN {X 0,Y 524.067,Z 565.203,A -85,B 0,C 180,E1 -4863.075,E2 -4863.075} C_VEL
LIN {X 0,Y 524.042,Z 565.198,A -85,B 0,C 180,E1 -4866.159,E2 -4866.159} C_VEL
LIN {X 0,Y 523.994,Z 565.212,A -85,B 0,C 180,E1 -4869.262,E2 -4869.262} C_VEL
LIN {X 0,Y 523.998,Z 565.204,A -85,B 0,C 180,E1 -4871.743,E2 -4871.743} C_VEL
LIN {X 0,Y 523.982,Z 565.218,A -85,B 0,C 180,E1 -4875.053,E2 -4875.053} C_VEL
LIN {X 0,Y 523.955,Z 565.211,A -85,B 0,C 180,E1 -4877.969,E2 -4877.969} C_VEL
LIN {X 0,Y 523.963,Z 565.212,A -85,B 0,C 180,E1 -4880.41,E2 -4880.41} C_VEL
LIN {X 0,Y 523.908,Z 565.227,A -85,B 0,C 180,E1 -4882.894,E2 -4882.894} C_VEL
LIN {X 0,Y 523.946,Z 565.218,A -85,B 0,C 180,E1 -4885.419,E2 -4885.419} C_VEL
LIN {X 0,Y 523.963,Z 565.213,A -85,B 0,C 180,E1 -4887.999,E2 -4887.999} C_VEL
LIN {X 0,Y 523.945,Z 565.217,A -85,B 0,C 180,E1 -4890.857,E2 -4890.857} C_VEL
LIN {X 0,Y 523.954,Z 565.213,A -85,B 0,C 180,E1 -4893.736,E2 -4893.736} C_VEL
LIN {X 0,Y 523.916,Z 565.219,A -85,B 0,C 180,E1 -4896.405,E2 -4896.405} C_VEL
LIN {X 0,Y 523.919,Z 565.226,A -85,B 0,C 180,E1 -4899.085,E2 -4899.085} C_VEL
LIN {X 0,Y 523.952,Z 565.206,A -85,B 0,C 180,E1 -4902.119,E2 -4902.119} C_VEL
LIN {X 0,Y 523.949,Z 565.224,A -85,B 0,C 180,E1 -4905.31,E2 -4905.31} C_VEL
LIN {X 0,Y 523.91,Z 565.22,A -85,B 0,C 180,E1 -4906.928,E2 -4906.928} C_VEL
LIN {X 0,Y 523.247,Z 565.303,A -85,B 0,C 180,E1 -4907.569,E2 -4907.569} C_VEL
LIN {X 0,Y 520.405,Z 565.656,A -85,B 0,C 180,E1 -4908.611,E2 -4908.611} C_VEL
LIN {X 0,Y 518,Z 565.964,A -85,B 0,C 180,E1 -4909.45,E2 -4909.45} C_VEL
LIN {X 0,Y 516.964,Z 566.087,A -85,B 0,C 180,E1 -4910.098,E2 -4910.098} C_VEL
LIN {X 0,Y 516.878,Z 566.096,A -85,B 0,C 180,E1 -4910.317,E2 -4910.317} C_VEL
LIN {X 0,Y 516.883,Z 566.101,A -85,B 0,C 180,E1 -4913.343,E2 -4913.343} C_VEL
LIN {X 0,Y 516.911,Z 566.093,A -85,B 0,C 180,E1 -4916.122,E2 -4916.122} C_VEL
LIN {X 0,Y 516.89,Z 566.096,A -85,B 0,C 180,E1 -4918.936,E2 -4918.936} C_VEL
LIN {X 0,Y 516.918,Z 566.099,A -85,B 0,C 180,E1 -4921.586,E2 -4921.586} C_VEL
LIN {X 0,Y 516.942,Z 566.093,A -85,B 0,C 180,E1 -4922.695,E2 -4922.695} C_VEL
LIN {X 0,Y 519.104,Z 576.487,A -85,B 0,C 180,E1 -4922.921,E2 -4922.921} C_VEL
LIN {X 0,Y 518.635,Z 670.844,A -85,B 0,C 180,E1 -4924.249,E2 -4924.249} C_VEL
LIN {X 0,Y 518.411,Z 684.253,A -85,B 0,C 180,E1 -4924.587,E2 -4924.587} C_VEL
LIN {X 0,Y 518.233,Z 697.083,A -85,B 0,C 180,E1 -4925.087,E2 -4925.087} C_VEL
LIN {X 0,Y 517.964,Z 709.155,A -85,B 0,C 180,E1 -4925.727,E2 -4925.727} C_VEL
LIN {X 0,Y 517.65,Z 720.409,A -85,B 0,C 180,E1 -4926.496,E2 -4926.496} C_VEL
LIN {X 0,Y 517.301,Z 730.993,A -85,B 0,C 180,E1 -4927.412,E2 -4927.412} C_VEL
LIN {X 0,Y 517.01,Z 740.83,A -85,B 0,C 180,E1 -4928.468,E2 -4928.468} C_VEL
LIN {X 0,Y 516.757,Z 749.26,A -85,B 0,C 180,E1 -4929.6,E2 -4929.6} C_VEL
LIN {X 0,Y 516.586,Z 756.126,A -85,B 0,C 180,E1 -4930.737,E2 -4930.737} C_VEL
LIN {X 0,Y 516.429,Z 762.604,A -85,B 0,C 180,E1 -4932.085,E2 -4932.085} C_VEL
LIN {X 0,Y 516.325,Z 767.338,A -85,B 0,C 180,E1 -4933.391,E2 -4933.391} C_VEL
LIN {X 0,Y 516.282,Z 769.629,A -85,B 0,C 180,E1 -4934.202,E2 -4934.202} C_VEL
LIN {X 0,Y 516.259,Z 771.695,A -85,B 0,C 180,E1 -4935.139,E2 -4935.139} C_VEL
LIN {X 0,Y 516.184,Z 773.759,A -85,B 0,C 180,E1 -4936.617,E2 -4936.617} C_VEL
LIN {X 0,Y 516.209,Z 774.302,A -85,B 0,C 180,E1 -4937.418,E2 -4937.418} C_VEL
LIN {X 0,Y 516.282,Z 774.325,A -85,B 0,C 180,E1 -4938.556,E2 -4938.556} C_VEL
LIN {X 0,Y 516.239,Z 773.422,A -85,B 0,C 180,E1 -4939.806,E2 -4939.806} C_VEL
LIN {X 0,Y 516.192,Z 772.33,A -85,B 0,C 180,E1 -4940.597,E2 -4940.597} C_VEL
LIN {X 0,Y 516.253,Z 770.798,A -85,B 0,C 180,E1 -4941.388,E2 -4941.388} C_VEL
LIN {X 0,Y 516.383,Z 767.71,A -85,B 0,C 180,E1 -4942.571,E2 -4942.571} C_VEL
LIN {X 0,Y 516.404,Z 763.604,A -85,B 0,C 180,E1 -4943.75,E2 -4943.75} C_VEL
LIN {X 0,Y 516.462,Z 758.356,A -85,B 0,C 180,E1 -4944.926,E2 -4944.926} C_VEL
LIN {X 0,Y 516.677,Z 751.782,A -85,B 0,C 180,E1 -4946.1,E2 -4946.1} C_VEL
LIN {X 0,Y 516.862,Z 743.599,A -85,B 0,C 180,E1 -4947.272,E2 -4947.272} C_VEL
LIN {X 0,Y 517.163,Z 735.208,A -85,B 0,C 180,E1 -4948.248,E2 -4948.248} C_VEL
LIN {X 0,Y 517.439,Z 724.981,A -85,B 0,C 180,E1 -4949.222,E2 -4949.222} C_VEL
LIN {X 0,Y 517.752,Z 714.799,A -85,B 0,C 180,E1 -4950,E2 -4950} C_VEL
LIN {X 0,Y 518.094,Z 703.537,A -85,B 0,C 180,E1 -4950.68,E2 -4950.68} C_VEL
LIN {X 0,Y 518.318,Z 690.966,A -85,B 0,C 180,E1 -4951.263,E2 -4951.263} C_VEL
LIN {X 0,Y 518.56,Z 678.214,A -85,B 0,C 180,E1 -4951.675,E2 -4951.675} C_VEL
LIN {X 0,Y 518.707,Z 664.766,A -85,B 0,C 180,E1 -4951.941,E2 -4951.941} C_VEL
LIN {X 0,Y 519.004,Z 574.31,A -85,B 0,C 180,E1 -4953.202,E2 -4953.202} C_VEL
LIN {X 0,Y 517.698,Z 568.426,A -85,B 0,C 180,E1 -4953.326,E2 -4953.326} C_VEL
LIN {X 0,Y 516.96,Z 566.092,A -85,B 0,C 180,E1 -4953.385,E2 -4953.385} C_VEL
LIN {X 0,Y 517.005,Z 566.087,A -85,B 0,C 180,E1 -4956.243,E2 -4956.243} C_VEL
LIN {X 0,Y 516.945,Z 566.089,A -85,B 0,C 180,E1 -4959.389,E2 -4959.389} C_VEL
LIN {X 0,Y 516.987,Z 566.088,A -85,B 0,C 180,E1 -4961.824,E2 -4961.824} C_VEL
LIN {X 0,Y 516.947,Z 566.087,A -85,B 0,C 180,E1 -4965.146,E2 -4965.146} C_VEL
LIN {X 0,Y 516.927,Z 566.096,A -85,B 0,C 180,E1 -4968.222,E2 -4968.222} C_VEL
LIN {X 0,Y 516.914,Z 566.091,A -85,B 0,C 180,E1 -4970.701,E2 -4970.701} C_VEL
LIN {X 0,Y 516.887,Z 566.103,A -85,B 0,C 180,E1 -4974.073,E2 -4974.073} C_VEL
LIN {X 0,Y 516.927,Z 566.092,A -85,B 0,C 180,E1 -4976.657,E2 -4976.657} C_VEL
LIN {X 0,Y 516.92,Z 566.095,A -85,B 0,C 180,E1 -4979.525,E2 -4979.525} C_VEL
LIN {X 0,Y 516.999,Z 566.088,A -85,B 0,C 180,E1 -4980.704,E2 -4980.704} C_VEL
LIN {X 0,Y 518.463,Z 571.645,A -85,B 0,C 180,E1 -4980.837,E2 -4980.837} C_VEL
LIN {X 0,Y 519.147,Z 576.346,A -85,B 0,C 180,E1 -4980.925,E2 -4980.925} C_VEL
LIN {X 0,Y 518.633,Z 670.732,A -85,B 0,C 180,E1 -4982.26,E2 -4982.26} C_VEL
LIN {X 0,Y 518.473,Z 681.872,A -85,B 0,C 180,E1 -4982.53,E2 -4982.53} C_VEL
LIN {X 0,Y 518.288,Z 693.968,A -85,B 0,C 180,E1 -4982.962,E2 -4982.962} C_VEL
LIN {X 0,Y 517.961,Z 707.263,A -85,B 0,C 180,E1 -4983.625,E2 -4983.625} C_VEL
LIN {X 0,Y 517.685,Z 717.554,A -85,B 0,C 180,E1 -4984.299,E2 -4984.299} C_VEL
LIN {X 0,Y 517.419,Z 726.26,A -85,B 0,C 180,E1 -4984.992,E2 -4984.992} C_VEL
LIN {X 0,Y 517.167,Z 735.396,A -85,B 0,C 180,E1 -4985.876,E2 -4985.876} C_VEL
LIN {X 0,Y 516.936,Z 742.863,A -85,B 0,C 180,E1 -4986.74,E2 -4986.74} C_VEL
LIN {X 0,Y 516.773,Z 748.409,A -85,B 0,C 180,E1 -4987.487,E2 -4987.487} C_VEL
LIN {X 0,Y 516.603,Z 754.837,A -85,B 0,C 180,E1 -4988.517,E2 -4988.517} C_VEL
LIN {X 0,Y 516.534,Z 759.554,A -85,B 0,C 180,E1 -4989.417,E2 -4989.417} C_VEL
LIN {X 0,Y 516.405,Z 763.649,A -85,B 0,C 180,E1 -4990.347,E2 -4990.347} C_VEL
LIN {X 0,Y 516.331,Z 767.754,A -85,B 0,C 180,E1 -4991.528,E2 -4991.528} C_VEL
LIN {X 0,Y 516.227,Z 771.18,A -85,B 0,C 180,E1 -4992.898,E2 -4992.898} C_VEL
LIN {X 0,Y 516.207,Z 773.015,A -85,B 0,C 180,E1 -4993.974,E2 -4993.974} C_VEL
LIN {X 0,Y 516.213,Z 774.102,A -85,B 0,C 180,E1 -4995.067,E2 -4995.067} C_VEL
LIN {X 0,Y 516.167,Z 774.421,A -85,B 0,C 180,E1 -4996.188,E2 -4996.188} C_VEL
LIN {X 0,Y 516.174,Z 773.914,A -85,B 0,C 180,E1 -4997.326,E2 -4997.326} C_VEL
LIN {X 0,Y 516.224,Z 772.539,A -85,B 0,C 180,E1 -4998.483,E2 -4998.483} C_VEL
LIN {X 0,Y 516.245,Z 770.194,A -85,B 0,C 180,E1 -4999.672,E2 -4999.672} C_VEL
LIN {X 0,Y 516.369,Z 765.49,A -85,B 0,C 180,E1 -5001.238,E2 -5001.238} C_VEL
LIN {X 0,Y 516.454,Z 761.539,A -85,B 0,C 180,E1 -5002.239,E2 -5002.239} C_VEL
LIN {X 0,Y 516.574,Z 755.907,A -85,B 0,C 180,E1 -5003.386,E2 -5003.386} C_VEL
LIN {X 0,Y 516.765,Z 749.272,A -85,B 0,C 180,E1 -5004.482,E2 -5004.482} C_VEL
LIN {X 0,Y 516.945,Z 742.544,A -85,B 0,C 180,E1 -5005.401,E2 -5005.401} C_VEL
LIN {X 0,Y 517.202,Z 733.991,A -85,B 0,C 180,E1 -5006.377,E2 -5006.377} C_VEL
LIN {X 0,Y 517.569,Z 722.442,A -85,B 0,C 180,E1 -5007.428,E2 -5007.428} C_VEL
LIN {X 0,Y 517.85,Z 712.515,A -85,B 0,C 180,E1 -5008.144,E2 -5008.144} C_VEL
LIN {X 0,Y 518.058,Z 702.692,A -85,B 0,C 180,E1 -5008.72,E2 -5008.72} C_VEL
LIN {X 0,Y 518.282,Z 692.058,A -85,B 0,C 180,E1 -5009.21,E2 -5009.21} C_VEL
LIN {X 0,Y 518.461,Z 680.566,A -85,B 0,C 180,E1 -5009.602,E2 -5009.602} C_VEL
LIN {X 0,Y 518.667,Z 668.026,A -85,B 0,C 180,E1 -5009.882,E2 -5009.882} C_VEL
LIN {X 0,Y 518.963,Z 575.711,A -85,B 0,C 180,E1 -5011.182,E2 -5011.182} C_VEL
LIN {X 0,Y 517.238,Z 567.559,A -85,B 0,C 180,E1 -5011.355,E2 -5011.355} C_VEL
LIN {X 0,Y 516.982,Z 566.58,A -85,B 0,C 180,E1 -5011.395,E2 -5011.395} C_VEL
LIN {X 0,Y 516.923,Z 566.097,A -85,B 0,C 180,E1 -5011.585,E2 -5011.585} C_VEL
LIN {X 0,Y 516.925,Z 566.097,A -85,B 0,C 180,E1 -5014.21,E2 -5014.21} C_VEL
LIN {X 0,Y 516.863,Z 566.105,A -85,B 0,C 180,E1 -5016.776,E2 -5016.776} C_VEL
LIN {X 0,Y 516.93,Z 566.091,A -85,B 0,C 180,E1 -5019.731,E2 -5019.731} C_VEL
LIN {X 0,Y 516.921,Z 566.099,A -85,B 0,C 180,E1 -5022.596,E2 -5022.596} C_VEL
LIN {X 0,Y 516.931,Z 566.093,A -85,B 0,C 180,E1 -5025.03,E2 -5025.03} C_VEL
LIN {X 0,Y 516.994,Z 566.087,A -85,B 0,C 180,E1 -5028.234,E2 -5028.234} C_VEL
LIN {X 0,Y 516.963,Z 566.086,A -85,B 0,C 180,E1 -5031.4,E2 -5031.4} C_VEL
LIN {X 0,Y 517.051,Z 566.082,A -85,B 0,C 180,E1 -5034.54,E2 -5034.54} C_VEL
LIN {X 0,Y 517.075,Z 566.07,A -85,B 0,C 180,E1 -5037.663,E2 -5037.663} C_VEL
LIN {X 0,Y 517.085,Z 566.075,A -85,B 0,C 180,E1 -5040.779,E2 -5040.779} C_VEL
LIN {X 0,Y 517.008,Z 566.079,A -85,B 0,C 180,E1 -5043.117,E2 -5043.117} C_VEL
LIN {X 0,Y 517.005,Z 566.085,A -85,B 0,C 180,E1 -5046.243,E2 -5046.243} C_VEL
LIN {X 0,Y 516.949,Z 566.085,A -85,B 0,C 180,E1 -5049.389,E2 -5049.389} C_VEL
LIN {X 0,Y 516.973,Z 566.083,A -85,B 0,C 180,E1 -5051.824,E2 -5051.824} C_VEL
LIN {X 0,Y 516.936,Z 566.088,A -85,B 0,C 180,E1 -5055.148,E2 -5055.148} C_VEL
LIN {X 0,Y 516.917,Z 566.093,A -85,B 0,C 180,E1 -5058.223,E2 -5058.223} C_VEL
LIN {X 0,Y 516.906,Z 566.097,A -85,B 0,C 180,E1 -5060.702,E2 -5060.702} C_VEL
LIN {X 0,Y 516.883,Z 566.094,A -85,B 0,C 180,E1 -5063.223,E2 -5063.223} C_VEL
LIN {X 0,Y 516.936,Z 566.093,A -85,B 0,C 180,E1 -5066.197,E2 -5066.197} C_VEL
LIN {X 0,Y 516.928,Z 566.09,A -85,B 0,C 180,E1 -5069.304,E2 -5069.304} C_VEL
LIN {X 0,Y 516.894,Z 566.101,A -85,B 0,C 180,E1 -5072.545,E2 -5072.545} C_VEL
LIN {X 0,Y 516.877,Z 566.096,A -85,B 0,C 180,E1 -5075.333,E2 -5075.333} C_VEL
LIN {X 0,Y 516.877,Z 566.098,A -85,B 0,C 180,E1 -5077.944,E2 -5077.944} C_VEL
LIN {X 0,Y 516.899,Z 566.098,A -85,B 0,C 180,E1 -5080.74,E2 -5080.74} C_VEL
LIN {X 0,Y 516.878,Z 566.097,A -85,B 0,C 180,E1 -5083.904,E2 -5083.904} C_VEL
LIN {X 0,Y 516.878,Z 566.1,A -85,B 0,C 180,E1 -5086.108,E2 -5086.108} C_VEL
LIN {X 0,Y 516.914,Z 566.099,A -85,B 0,C 180,E1 -5088.399,E2 -5088.399} C_VEL
LIN {X 0,Y 516.884,Z 566.096,A -85,B 0,C 180,E1 -5091.286,E2 -5091.286} C_VEL
LIN {X 0,Y 516.874,Z 566.102,A -85,B 0,C 180,E1 -5094.221,E2 -5094.221} C_VEL
LIN {X 0,Y 516.895,Z 566.097,A -85,B 0,C 180,E1 -5097.054,E2 -5097.054} C_VEL
LIN {X 0,Y 516.891,Z 566.097,A -85,B 0,C 180,E1 -5099.797,E2 -5099.797} C_VEL
LIN {X 0,Y 516.923,Z 566.098,A -85,B 0,C 180,E1 -5102.906,E2 -5102.906} C_VEL
LIN {X 0,Y 516.965,Z 566.194,A -85,B 0,C 180,E1 -5103.182,E2 -5103.182} C_VEL
LIN {X 0,Y 519.089,Z 577.014,A -85,B 0,C 180,E1 -5104.799,E2 -5104.799} C_VEL
LIN {X 0,Y 518.697,Z 594.606,A -85,B 0,C 180,E1 -5107.228,E2 -5107.228} C_VEL
LIN {X 0,Y 518.198,Z 617.922,A -85,B 0,C 180,E1 -5110.387,E2 -5110.387} C_VEL
LIN {X 0,Y 517.605,Z 643.664,A -85,B 0,C 180,E1 -5113.839,E2 -5113.839} C_VEL
LIN {X 0,Y 517.514,Z 649.538,A -85,B 0,C 180,E1 -5114.624,E2 -5114.624} C_VEL
LIN {X 0,Y 519.07,Z 661.845,A -85,B 0,C 180,E1 -5114.849,E2 -5114.849} C_VEL
LIN {X 0,Y 518.672,Z 758.659,A -85,B 0,C 180,E1 -5116.209,E2 -5116.209} C_VEL
LIN {X 0,Y 518.385,Z 771.355,A -85,B 0,C 180,E1 -5116.525,E2 -5116.525} C_VEL
LIN {X 0,Y 518.153,Z 784.43,A -85,B 0,C 180,E1 -5117.018,E2 -5117.018} C_VEL
LIN {X 0,Y 517.877,Z 795.977,A -85,B 0,C 180,E1 -5117.606,E2 -5117.606} C_VEL
LIN {X 0,Y 517.585,Z 807.278,A -85,B 0,C 180,E1 -5118.348,E2 -5118.348} C_VEL
LIN {X 0,Y 517.262,Z 818.056,A -85,B 0,C 180,E1 -5119.233,E2 -5119.233} C_VEL
LIN {X 0,Y 517.02,Z 827.784,A -85,B 0,C 180,E1 -5120.217,E2 -5120.217} C_VEL
LIN {X 0,Y 516.775,Z 835.759,A -85,B 0,C 180,E1 -5121.2,E2 -5121.2} C_VEL
LIN {X 0,Y 516.563,Z 843.552,A -85,B 0,C 180,E1 -5122.377,E2 -5122.377} C_VEL
LIN {X 0,Y 516.43,Z 849.227,A -85,B 0,C 180,E1 -5123.437,E2 -5123.437} C_VEL
LIN {X 0,Y 516.405,Z 853.948,A -85,B 0,C 180,E1 -5124.533,E2 -5124.533} C_VEL
LIN {X 0,Y 516.344,Z 857.895,A -85,B 0,C 180,E1 -5125.707,E2 -5125.707} C_VEL
LIN {X 0,Y 516.282,Z 860.81,A -85,B 0,C 180,E1 -5126.879,E2 -5126.879} C_VEL
LIN {X 0,Y 516.26,Z 862.195,A -85,B 0,C 180,E1 -5127.659,E2 -5127.659} C_VEL
LIN {X 0,Y 516.16,Z 863.786,A -85,B 0,C 180,E1 -5129.22,E2 -5129.22} C_VEL
LIN {X 0,Y 516.154,Z 864,A -85,B 0,C 180,E1 -5130,E2 -5130} C_VEL
LIN {X 0,Y 516.191,Z 863.181,A -85,B 0,C 180,E1 -5131.56,E2 -5131.56} C_VEL
LIN {X 0,Y 516.26,Z 862.193,A -85,B 0,C 180,E1 -5132.341,E2 -5132.341} C_VEL
LIN {X 0,Y 516.282,Z 860.807,A -85,B 0,C 180,E1 -5133.121,E2 -5133.121} C_VEL
LIN {X 0,Y 516.344,Z 857.894,A -85,B 0,C 180,E1 -5134.293,E2 -5134.293} C_VEL
LIN {X 0,Y 516.405,Z 853.95,A -85,B 0,C 180,E1 -5135.467,E2 -5135.467} C_VEL
LIN {X 0,Y 516.486,Z 848.016,A -85,B 0,C 180,E1 -5136.807,E2 -5136.807} C_VEL
LIN {X 0,Y 516.64,Z 841.127,A -85,B 0,C 180,E1 -5138.015,E2 -5138.015} C_VEL
LIN {X 0,Y 516.844,Z 832.756,A -85,B 0,C 180,E1 -5139.194,E2 -5139.194} C_VEL
LIN {X 0,Y 517.069,Z 824.179,A -85,B 0,C 180,E1 -5140.177,E2 -5140.177} C_VEL
LIN {X 0,Y 517.433,Z 813.598,A -85,B 0,C 180,E1 -5141.16,E2 -5141.16} C_VEL
LIN {X 0,Y 517.668,Z 801.968,A -85,B 0,C 180,E1 -5142.028,E2 -5142.028} C_VEL
LIN {X 0,Y 518.036,Z 789.717,A -85,B 0,C 180,E1 -5142.736,E2 -5142.736} C_VEL
LIN {X 0,Y 518.318,Z 777.275,A -85,B 0,C 180,E1 -5143.277,E2 -5143.277} C_VEL
LIN {X 0,Y 518.547,Z 764.48,A -85,B 0,C 180,E1 -5143.67,E2 -5143.67} C_VEL
LIN {X 0,Y 518.739,Z 749.287,A -85,B 0,C 180,E1 -5143.94,E2 -5143.94} C_VEL
LIN {X 0,Y 518.993,Z 658.588,A -85,B 0,C 180,E1 -5145.201,E2 -5145.201} C_VEL
LIN {X 0,Y 517.714,Z 648.815,A -85,B 0,C 180,E1 -5145.384,E2 -5145.384} C_VEL
LIN {X 0,Y 518.293,Z 621.487,A -85,B 0,C 180,E1 -5148.597,E2 -5148.597} C_VEL
LIN {X 0,Y 518.987,Z 595.701,A -85,B 0,C 180,E1 -5151.654,E2 -5151.654} C_VEL
LIN {X 0,Y 519.401,Z 578.396,A -85,B 0,C 180,E1 -5153.737,E2 -5153.737} C_VEL
LIN {X 0,Y 518.383,Z 572.649,A -85,B 0,C 180,E1 -5154.488,E2 -5154.488} C_VEL
LIN {X 0,Y 516.941,Z 566.095,A -85,B 0,C 180,E1 -5155.383,E2 -5155.383} C_VEL
LIN {X 0,Y 516.92,Z 566.094,A -85,B 0,C 180,E1 -5158.414,E2 -5158.414} C_VEL
LIN {X 0,Y 516.888,Z 566.096,A -85,B 0,C 180,E1 -5161.109,E2 -5161.109} C_VEL
LIN {X 0,Y 516.913,Z 566.1,A -85,B 0,C 180,E1 -5163.966,E2 -5163.966} C_VEL
LIN {X 0,Y 516.881,Z 566.096,A -85,B 0,C 180,E1 -5166.745,E2 -5166.745} C_VEL
LIN {X 0,Y 516.9,Z 566.096,A -85,B 0,C 180,E1 -5169.718,E2 -5169.718} C_VEL
LIN {X 0,Y 516.915,Z 566.095,A -85,B 0,C 180,E1 -5171.774,E2 -5171.774} C_VEL
LIN {X 0,Y 516.918,Z 566.089,A -85,B 0,C 180,E1 -5175.009,E2 -5175.009} C_VEL
LIN {X 0,Y 516.919,Z 566.095,A -85,B 0,C 180,E1 -5178.397,E2 -5178.397} C_VEL
LIN {X 0,Y 516.901,Z 566.091,A -85,B 0,C 180,E1 -5181.286,E2 -5181.286} C_VEL
LIN {X 0,Y 516.885,Z 566.1,A -85,B 0,C 180,E1 -5184.221,E2 -5184.221} C_VEL
LIN {X 0,Y 516.89,Z 566.094,A -85,B 0,C 180,E1 -5187.053,E2 -5187.053} C_VEL
LIN {X 0,Y 516.894,Z 566.094,A -85,B 0,C 180,E1 -5189.796,E2 -5189.796} C_VEL
LIN {X 0,Y 516.922,Z 566.097,A -85,B 0,C 180,E1 -5192.467,E2 -5192.467} C_VEL
LIN {X 0,Y 516.903,Z 566.092,A -85,B 0,C 180,E1 -5195.071,E2 -5195.071} C_VEL
LIN {X 0,Y 516.878,Z 566.099,A -85,B 0,C 180,E1 -5198.462,E2 -5198.462} C_VEL
LIN {X 0,Y 516.896,Z 566.095,A -85,B 0,C 180,E1 -5200.955,E2 -5200.955} C_VEL
LIN {X 0,Y 516.907,Z 566.087,A -85,B 0,C 180,E1 -5203.41,E2 -5203.41} C_VEL
LIN {X 0,Y 516.885,Z 566.093,A -85,B 0,C 180,E1 -5205.833,E2 -5205.833} C_VEL
LIN {X 0,Y 516.948,Z 566.087,A -85,B 0,C 180,E1 -5209.028,E2 -5209.028} C_VEL
LIN {X 0,Y 516.969,Z 566.081,A -85,B 0,C 180,E1 -5212.187,E2 -5212.187} C_VEL
LIN {X 0,Y 517.055,Z 566.08,A -85,B 0,C 180,E1 -5214.54,E2 -5214.54} C_VEL
LIN {X 0,Y 517.075,Z 566.066,A -85,B 0,C 180,E1 -5217.663,E2 -5217.663} C_VEL
LIN {X 0,Y 517.087,Z 566.077,A -85,B 0,C 180,E1 -5220.779,E2 -5220.779} C_VEL
LIN {X 0,Y 517.007,Z 566.082,A -85,B 0,C 180,E1 -5223.117,E2 -5223.117} C_VEL
LIN {X 0,Y 517.005,Z 566.075,A -85,B 0,C 180,E1 -5226.243,E2 -5226.243} C_VEL
LIN {X 0,Y 516.948,Z 566.088,A -85,B 0,C 180,E1 -5229.389,E2 -5229.389} C_VEL
LIN {X 0,Y 516.947,Z 566.082,A -85,B 0,C 180,E1 -5231.811,E2 -5231.811} C_VEL
LIN {X 0,Y 516.934,Z 566.094,A -85,B 0,C 180,E1 -5235.147,E2 -5235.147} C_VEL
LIN {X 0,Y 516.916,Z 566.088,A -85,B 0,C 180,E1 -5238.223,E2 -5238.223} C_VEL
LIN {X 0,Y 516.904,Z 566.095,A -85,B 0,C 180,E1 -5240.702,E2 -5240.702} C_VEL
LIN {X 0,Y 516.902,Z 566.089,A -85,B 0,C 180,E1 -5244.073,E2 -5244.073} C_VEL
LIN {X 0,Y 516.921,Z 566.092,A -85,B 0,C 180,E1 -5246.658,E2 -5246.658} C_VEL
LIN {X 0,Y 516.917,Z 566.09,A -85,B 0,C 180,E1 -5249.527,E2 -5249.527} C_VEL
LIN {X 0,Y 516.893,Z 566.095,A -85,B 0,C 180,E1 -5252.545,E2 -5252.545} C_VEL
LIN {X 0,Y 516.876,Z 566.103,A -85,B 0,C 180,E1 -5255.333,E2 -5255.333} C_VEL
LIN {X 0,Y 516.879,Z 566.096,A -85,B 0,C 180,E1 -5257.945,E2 -5257.945} C_VEL
LIN {X 0,Y 516.88,Z 566.096,A -85,B 0,C 180,E1 -5260.742,E2 -5260.742} C_VEL
LIN {X 0,Y 516.9,Z 566.086,A -85,B 0,C 180,E1 -5262.83,E2 -5262.83} C_VEL
LIN {X 0,Y 516.918,Z 566.095,A -85,B 0,C 180,E1 -5265.011,E2 -5265.011} C_VEL
LIN {X 0,Y 516.911,Z 566.088,A -85,B 0,C 180,E1 -5268.399,E2 -5268.399} C_VEL
LIN {X 0,Y 516.878,Z 566.096,A -85,B 0,C 180,E1 -5270.317,E2 -5270.317} C_VEL
LIN {X 0,Y 516.21,Z 566.184,A -85,B 0,C 180,E1 -5270.967,E2 -5270.967} C_VEL
LIN {X 0,Y 513.364,Z 566.542,A -85,B 0,C 180,E1 -5272.023,E2 -5272.023} C_VEL
LIN {X 0,Y 510.956,Z 566.844,A -85,B 0,C 180,E1 -5272.874,E2 -5272.874} C_VEL
LIN {X 0,Y 509.917,Z 566.971,A -85,B 0,C 180,E1 -5273.53,E2 -5273.53} C_VEL
LIN {X 0,Y 509.829,Z 566.978,A -85,B 0,C 180,E1 -5273.752,E2 -5273.752} C_VEL
LIN {X 0,Y 509.86,Z 566.971,A -85,B 0,C 180,E1 -5276.54,E2 -5276.54} C_VEL
LIN {X 0,Y 509.844,Z 566.979,A -85,B 0,C 180,E1 -5279.335,E2 -5279.335} C_VEL
LIN {X 0,Y 509.906,Z 567.021,A -85,B 0,C 180,E1 -5282.496,E2 -5282.496} C_VEL
LIN {X 0,Y 512.021,Z 575.829,A -85,B 0,C 180,E1 -5282.69,E2 -5282.69} C_VEL
LIN {X 0,Y 512.253,Z 579.451,A -85,B 0,C 180,E1 -5282.749,E2 -5282.749} C_VEL
LIN {X 0,Y 511.757,Z 671.782,A -85,B 0,C 180,E1 -5284.068,E2 -5284.068} C_VEL
LIN {X 0,Y 511.534,Z 685.089,A -85,B 0,C 180,E1 -5284.411,E2 -5284.411} C_VEL
LIN {X 0,Y 511.354,Z 697.45,A -85,B 0,C 180,E1 -5284.9,E2 -5284.9} C_VEL
LIN {X 0,Y 511.06,Z 709.895,A -85,B 0,C 180,E1 -5285.567,E2 -5285.567} C_VEL
LIN {X 0,Y 510.744,Z 720.083,A -85,B 0,C 180,E1 -5286.267,E2 -5286.267} C_VEL
LIN {X 0,Y 510.382,Z 729.978,A -85,B 0,C 180,E1 -5287.108,E2 -5287.108} C_VEL
LIN {X 0,Y 510.095,Z 739.935,A -85,B 0,C 180,E1 -5288.162,E2 -5288.162} C_VEL
LIN {X 0,Y 509.829,Z 747.863,A -85,B 0,C 180,E1 -5289.189,E2 -5289.189} C_VEL
LIN {X 0,Y 509.615,Z 754.626,A -85,B 0,C 180,E1 -5290.253,E2 -5290.253} C_VEL
LIN {X 0,Y 509.489,Z 761.028,A -85,B 0,C 180,E1 -5291.503,E2 -5291.503} C_VEL
LIN {X 0,Y 509.36,Z 766.014,A -85,B 0,C 180,E1 -5292.744,E2 -5292.744} C_VEL
LIN {X 0,Y 509.247,Z 769.792,A -85,B 0,C 180,E1 -5293.978,E2 -5293.978} C_VEL
LIN {X 0,Y 509.2,Z 772.212,A -85,B 0,C 180,E1 -5295.049,E2 -5295.049} C_VEL
LIN {X 0,Y 509.118,Z 774.197,A -85,B 0,C 180,E1 -5296.428,E2 -5296.428} C_VEL
LIN {X 0,Y 509.123,Z 774.812,A -85,B 0,C 180,E1 -5297.24,E2 -5297.24} C_VEL
LIN {X 0,Y 509.209,Z 774.939,A -85,B 0,C 180,E1 -5298.502,E2 -5298.502} C_VEL
LIN {X 0,Y 509.177,Z 774.185,A -85,B 0,C 180,E1 -5299.663,E2 -5299.663} C_VEL
LIN {X 0,Y 509.126,Z 773.194,A -85,B 0,C 180,E1 -5300.465,E2 -5300.465} C_VEL
LIN {X 0,Y 509.199,Z 771.756,A -85,B 0,C 180,E1 -5301.268,E2 -5301.268} C_VEL
LIN {X 0,Y 509.317,Z 768.808,A -85,B 0,C 180,E1 -5302.468,E2 -5302.468} C_VEL
LIN {X 0,Y 509.387,Z 764.84,A -85,B 0,C 180,E1 -5303.663,E2 -5303.663} C_VEL
LIN {X 0,Y 509.444,Z 759.749,A -85,B 0,C 180,E1 -5304.855,E2 -5304.855} C_VEL
LIN {X 0,Y 509.649,Z 753.352,A -85,B 0,C 180,E1 -5306.046,E2 -5306.046} C_VEL
LIN {X 0,Y 509.842,Z 745.449,A -85,B 0,C 180,E1 -5307.235,E2 -5307.235} C_VEL
LIN {X 0,Y 510.151,Z 737.33,A -85,B 0,C 180,E1 -5308.224,E2 -5308.224} C_VEL
LIN {X 0,Y 510.457,Z 727.396,A -85,B 0,C 180,E1 -5309.211,E2 -5309.211} C_VEL
LIN {X 0,Y 510.697,Z 717.672,A -85,B 0,C 180,E1 -5310,E2 -5310} C_VEL
LIN {X 0,Y 511.121,Z 707.053,A -85,B 0,C 180,E1 -5310.689,E2 -5310.689} C_VEL
LIN {X 0,Y 511.399,Z 695.415,A -85,B 0,C 180,E1 -5311.28,E2 -5311.28} C_VEL
LIN {X 0,Y 511.601,Z 682.768,A -85,B 0,C 180,E1 -5311.747,E2 -5311.747} C_VEL
LIN {X 0,Y 511.835,Z 669.412,A -85,B 0,C 180,E1 -5312.066,E2 -5312.066} C_VEL
LIN {X 0,Y 512.185,Z 575.067,A -85,B 0,C 180,E1 -5313.405,E2 -5313.405} C_VEL
LIN {X 0,Y 511.096,Z 570.753,A -85,B 0,C 180,E1 -5313.501,E2 -5313.501} C_VEL
LIN {X 0,Y 509.902,Z 566.972,A -85,B 0,C 180,E1 -5313.605,E2 -5313.605} C_VEL
LIN {X 0,Y 509.957,Z 566.964,A -85,B 0,C 180,E1 -5316.33,E2 -5316.33} C_VEL
LIN {X 0,Y 509.907,Z 566.966,A -85,B 0,C 180,E1 -5318.72,E2 -5318.72} C_VEL
LIN {X 0,Y 509.954,Z 566.965,A -85,B 0,C 180,E1 -5321.93,E2 -5321.93} C_VEL
LIN {X 0,Y 509.896,Z 566.966,A -85,B 0,C 180,E1 -5325.241,E2 -5325.241} C_VEL
LIN {X 0,Y 509.89,Z 566.974,A -85,B 0,C 180,E1 -5328,E2 -5328} C_VEL
LIN {X 0,Y 509.852,Z 566.97,A -85,B 0,C 180,E1 -5331.001,E2 -5331.001} C_VEL
LIN {X 0,Y 509.824,Z 566.977,A -85,B 0,C 180,E1 -5333.563,E2 -5333.563} C_VEL
LIN {X 0,Y 509.912,Z 566.969,A -85,B 0,C 180,E1 -5336.378,E2 -5336.378} C_VEL
LIN {X 0,Y 509.88,Z 566.971,A -85,B 0,C 180,E1 -5338.843,E2 -5338.843} C_VEL
LIN {X 0,Y 509.927,Z 566.969,A -85,B 0,C 180,E1 -5340.488,E2 -5340.488} C_VEL
LIN {X 0,Y 511.878,Z 573.9,A -85,B 0,C 180,E1 -5340.662,E2 -5340.662} C_VEL
LIN {X 0,Y 512.337,Z 578.049,A -85,B 0,C 180,E1 -5340.738,E2 -5340.738} C_VEL
LIN {X 0,Y 511.745,Z 671.47,A -85,B 0,C 180,E1 -5342.078,E2 -5342.078} C_VEL
LIN {X 0,Y 511.551,Z 684.126,A -85,B 0,C 180,E1 -5342.398,E2 -5342.398} C_VEL
LIN {X 0,Y 511.315,Z 697.878,A -85,B 0,C 180,E1 -5342.934,E2 -5342.934} C_VEL
LIN {X 0,Y 511.043,Z 708.339,A -85,B 0,C 180,E1 -5343.49,E2 -5343.49} C_VEL
LIN {X 0,Y 510.715,Z 719.648,A -85,B 0,C 180,E1 -5344.258,E2 -5344.258} C_VEL
LIN {X 0,Y 510.457,Z 728.157,A -85,B 0,C 180,E1 -5344.965,E2 -5344.965} C_VEL
LIN {X 0,Y 510.194,Z 736.141,A -85,B 0,C 180,E1 -5345.756,E2 -5345.756} C_VEL
LIN {X 0,Y 509.926,Z 744.695,A -85,B 0,C 180,E1 -5346.776,E2 -5346.776} C_VEL
LIN {X 0,Y 509.648,Z 752.865,A -85,B 0,C 180,E1 -5347.969,E2 -5347.969} C_VEL
LIN {X 0,Y 509.487,Z 760.408,A -85,B 0,C 180,E1 -5349.384,E2 -5349.384} C_VEL
LIN {X 0,Y 509.33,Z 765.539,A -85,B 0,C 180,E1 -5350.631,E2 -5350.631} C_VEL
LIN {X 0,Y 509.273,Z 769.316,A -85,B 0,C 180,E1 -5351.823,E2 -5351.823} C_VEL
LIN {X 0,Y 509.154,Z 772.034,A -85,B 0,C 180,E1 -5352.981,E2 -5352.981} C_VEL
LIN {X 0,Y 509.145,Z 773.839,A -85,B 0,C 180,E1 -5354.128,E2 -5354.128} C_VEL
LIN {X 0,Y 509.124,Z 774.802,A -85,B 0,C 180,E1 -5355.25,E2 -5355.25} C_VEL
LIN {X 0,Y 509.095,Z 774.994,A -85,B 0,C 180,E1 -5356.35,E2 -5356.35} C_VEL
LIN {X 0,Y 509.118,Z 774.443,A -85,B 0,C 180,E1 -5357.436,E2 -5357.436} C_VEL
LIN {X 0,Y 509.156,Z 773.182,A -85,B 0,C 180,E1 -5358.505,E2 -5358.505} C_VEL
LIN {X 0,Y 509.183,Z 771.198,A -85,B 0,C 180,E1 -5359.555,E2 -5359.555} C_VEL
LIN {X 0,Y 509.272,Z 768.464,A -85,B 0,C 180,E1 -5360.605,E2 -5360.605} C_VEL
LIN {X 0,Y 509.368,Z 764.172,A -85,B 0,C 180,E1 -5361.854,E2 -5361.854} C_VEL
LIN {X 0,Y 509.485,Z 758.434,A -85,B 0,C 180,E1 -5363.135,E2 -5363.135} C_VEL
LIN {X 0,Y 509.723,Z 751.894,A -85,B 0,C 180,E1 -5364.289,E2 -5364.289} C_VEL
LIN {X 0,Y 509.918,Z 744.536,A -85,B 0,C 180,E1 -5365.352,E2 -5365.352} C_VEL
LIN {X 0,Y 510.197,Z 736.351,A -85,B 0,C 180,E1 -5366.327,E2 -5366.327} C_VEL
LIN {X 0,Y 510.492,Z 727.252,A -85,B 0,C 180,E1 -5367.223,E2 -5367.223} C_VEL
LIN {X 0,Y 510.871,Z 715.736,A -85,B 0,C 180,E1 -5368.135,E2 -5368.135} C_VEL
LIN {X 0,Y 511.141,Z 704.17,A -85,B 0,C 180,E1 -5368.847,E2 -5368.847} C_VEL
LIN {X 0,Y 511.389,Z 692.856,A -85,B 0,C 180,E1 -5369.379,E2 -5369.379} C_VEL
LIN {X 0,Y 511.589,Z 681.583,A -85,B 0,C 180,E1 -5369.772,E2 -5369.772} C_VEL
LIN {X 0,Y 511.748,Z 669.459,A -85,B 0,C 180,E1 -5370.054,E2 -5370.054} C_VEL
LIN {X 0,Y 512.147,Z 576.429,A -85,B 0,C 180,E1 -5371.387,E2 -5371.387} C_VEL
LIN {X 0,Y 510.567,Z 569.301,A -85,B 0,C 180,E1 -5371.543,E2 -5371.543} C_VEL
LIN {X 0,Y 509.93,Z 567.143,A -85,B 0,C 180,E1 -5371.62,E2 -5371.62} C_VEL
LIN {X 0,Y 509.87,Z 566.976,A -85,B 0,C 180,E1 -5374.703,E2 -5374.703} C_VEL
LIN {X 0,Y 509.827,Z 566.976,A -85,B 0,C 180,E1 -5377.455,E2 -5377.455} C_VEL
LIN {X 0,Y 509.908,Z 566.966,A -85,B 0,C 180,E1 -5379.844,E2 -5379.844} C_VEL
LIN {X 0,Y 509.877,Z 566.97,A -85,B 0,C 180,E1 -5383.174,E2 -5383.174} C_VEL
LIN {X 0,Y 509.854,Z 566.972,A -85,B 0,C 180,E1 -5385.634,E2 -5385.634} C_VEL
LIN {X 0,Y 509.916,Z 566.968,A -85,B 0,C 180,E1 -5388.875,E2 -5388.875} C_VEL
LIN {X 0,Y 509.942,Z 566.963,A -85,B 0,C 180,E1 -5392.078,E2 -5392.078} C_VEL
LIN {X 0,Y 509.998,Z 566.961,A -85,B 0,C 180,E1 -5394.464,E2 -5394.464} C_VEL
LIN {X 0,Y 510.046,Z 566.946,A -85,B 0,C 180,E1 -5397.631,E2 -5397.631} C_VEL
LIN {X 0,Y 510.055,Z 566.951,A -85,B 0,C 180,E1 -5400.79,E2 -5400.79} C_VEL
LIN {X 0,Y 509.95,Z 566.958,A -85,B 0,C 180,E1 -5403.16,E2 -5403.16} C_VEL
LIN {X 0,Y 509.972,Z 566.962,A -85,B 0,C 180,E1 -5406.33,E2 -5406.33} C_VEL
LIN {X 0,Y 509.909,Z 566.968,A -85,B 0,C 180,E1 -5408.72,E2 -5408.72} C_VEL
LIN {X 0,Y 509.941,Z 566.96,A -85,B 0,C 180,E1 -5411.931,E2 -5411.931} C_VEL
LIN {X 0,Y 509.883,Z 566.966,A -85,B 0,C 180,E1 -5415.242,E2 -5415.242} C_VEL
LIN {X 0,Y 509.879,Z 566.967,A -85,B 0,C 180,E1 -5418.002,E2 -5418.002} C_VEL
LIN {X 0,Y 509.848,Z 566.973,A -85,B 0,C 180,E1 -5421.002,E2 -5421.002} C_VEL
LIN {X 0,Y 509.842,Z 566.97,A -85,B 0,C 180,E1 -5423.563,E2 -5423.563} C_VEL
LIN {X 0,Y 509.905,Z 566.972,A -85,B 0,C 180,E1 -5426.38,E2 -5426.38} C_VEL
LIN {X 0,Y 509.878,Z 566.972,A -85,B 0,C 180,E1 -5428.844,E2 -5428.844} C_VEL
LIN {X 0,Y 509.819,Z 566.975,A -85,B 0,C 180,E1 -5431.59,E2 -5431.59} C_VEL
LIN {X 0,Y 509.848,Z 566.977,A -85,B 0,C 180,E1 -5434.414,E2 -5434.414} C_VEL
LIN {X 0,Y 509.814,Z 566.976,A -85,B 0,C 180,E1 -5437.341,E2 -5437.341} C_VEL
LIN {X 0,Y 509.856,Z 566.977,A -85,B 0,C 180,E1 -5440.381,E2 -5440.381} C_VEL
LIN {X 0,Y 509.835,Z 566.975,A -85,B 0,C 180,E1 -5443.065,E2 -5443.065} C_VEL
LIN {X 0,Y 509.826,Z 566.976,A -85,B 0,C 180,E1 -5445.793,E2 -5445.793} C_VEL
LIN {X 0,Y 509.855,Z 566.979,A -85,B 0,C 180,E1 -5448.576,E2 -5448.576} C_VEL
LIN {X 0,Y 509.849,Z 566.973,A -85,B 0,C 180,E1 -5451.787,E2 -5451.787} C_VEL
LIN {X 0,Y 509.834,Z 566.98,A -85,B 0,C 180,E1 -5454.623,E2 -5454.623} C_VEL
LIN {X 0,Y 509.862,Z 566.972,A -85,B 0,C 180,E1 -5457.482,E2 -5457.482} C_VEL
LIN {X 0,Y 509.858,Z 566.977,A -85,B 0,C 180,E1 -5460.274,E2 -5460.274} C_VEL
LIN {X 0,Y 509.905,Z 567.003,A -85,B 0,C 180,E1 -5462.989,E2 -5462.989} C_VEL
LIN {X 0,Y 512.178,Z 579.139,A -85,B 0,C 180,E1 -5464.826,E2 -5464.826} C_VEL
LIN {X 0,Y 511.703,Z 596.216,A -85,B 0,C 180,E1 -5467.217,E2 -5467.217} C_VEL
LIN {X 0,Y 511.199,Z 618.762,A -85,B 0,C 180,E1 -5470.317,E2 -5470.317} C_VEL
LIN {X 0,Y 510.565,Z 644.471,A -85,B 0,C 180,E1 -5473.815,E2 -5473.815} C_VEL
LIN {X 0,Y 510.468,Z 648.91,A -85,B 0,C 180,E1 -5474.415,E2 -5474.415} C_VEL
LIN {X 0,Y 512.201,Z 662.469,A -85,B 0,C 180,E1 -5474.661,E2 -5474.661} C_VEL
LIN {X 0,Y 511.759,Z 758.888,A -85,B 0,C 180,E1 -5476.044,E2 -5476.044} C_VEL
LIN {X 0,Y 511.429,Z 772.035,A -85,B 0,C 180,E1 -5476.389,E2 -5476.389} C_VEL
LIN {X 0,Y 511.184,Z 784.766,A -85,B 0,C 180,E1 -5476.889,E2 -5476.889} C_VEL
LIN {X 0,Y 510.863,Z 796.271,A -85,B 0,C 180,E1 -5477.497,E2 -5477.497} C_VEL
LIN {X 0,Y 510.537,Z 807.844,A -85,B 0,C 180,E1 -5478.285,E2 -5478.285} C_VEL
LIN {X 0,Y 510.195,Z 818.42,A -85,B 0,C 180,E1 -5479.182,E2 -5479.182} C_VEL
LIN {X 0,Y 509.948,Z 827.08,A -85,B 0,C 180,E1 -5480.08,E2 -5480.08} C_VEL
LIN {X 0,Y 509.713,Z 835.072,A -85,B 0,C 180,E1 -5481.077,E2 -5481.077} C_VEL
LIN {X 0,Y 509.494,Z 842.883,A -85,B 0,C 180,E1 -5482.271,E2 -5482.271} C_VEL
LIN {X 0,Y 509.332,Z 849.14,A -85,B 0,C 180,E1 -5483.46,E2 -5483.46} C_VEL
LIN {X 0,Y 509.344,Z 853.428,A -85,B 0,C 180,E1 -5484.457,E2 -5484.457} C_VEL
LIN {X 0,Y 509.233,Z 857.455,A -85,B 0,C 180,E1 -5485.647,E2 -5485.647} C_VEL
LIN {X 0,Y 509.201,Z 860.435,A -85,B 0,C 180,E1 -5486.835,E2 -5486.835} C_VEL
LIN {X 0,Y 509.189,Z 861.852,A -85,B 0,C 180,E1 -5487.627,E2 -5487.627} C_VEL
LIN {X 0,Y 509.073,Z 863.469,A -85,B 0,C 180,E1 -5489.209,E2 -5489.209} C_VEL
LIN {X 0,Y 509.065,Z 863.689,A -85,B 0,C 180,E1 -5490,E2 -5490} C_VEL
LIN {X 0,Y 509.112,Z 862.857,A -85,B 0,C 180,E1 -5491.582,E2 -5491.582} C_VEL
LIN {X 0,Y 509.189,Z 861.854,A -85,B 0,C 180,E1 -5492.373,E2 -5492.373} C_VEL
LIN {X 0,Y 509.201,Z 860.439,A -85,B 0,C 180,E1 -5493.165,E2 -5493.165} C_VEL
LIN {X 0,Y 509.232,Z 857.468,A -85,B 0,C 180,E1 -5494.353,E2 -5494.353} C_VEL
LIN {X 0,Y 509.344,Z 853.451,A -85,B 0,C 180,E1 -5495.543,E2 -5495.543} C_VEL
LIN {X 0,Y 509.405,Z 847.716,A -85,B 0,C 180,E1 -5496.844,E2 -5496.844} C_VEL
LIN {X 0,Y 509.572,Z 840.499,A -85,B 0,C 180,E1 -5498.127,E2 -5498.127} C_VEL
LIN {X 0,Y 509.793,Z 832.121,A -85,B 0,C 180,E1 -5499.322,E2 -5499.322} C_VEL
LIN {X 0,Y 510.035,Z 823.533,A -85,B 0,C 180,E1 -5500.319,E2 -5500.319} C_VEL
LIN {X 0,Y 510.416,Z 812.94,A -85,B 0,C 180,E1 -5501.315,E2 -5501.315} C_VEL
LIN {X 0,Y 510.657,Z 801.295,A -85,B 0,C 180,E1 -5502.196,E2 -5502.196} C_VEL
LIN {X 0,Y 511.023,Z 790.976,A -85,B 0,C 180,E1 -5502.812,E2 -5502.812} C_VEL
LIN {X 0,Y 511.357,Z 779.165,A -85,B 0,C 180,E1 -5503.36,E2 -5503.36} C_VEL
LIN {X 0,Y 511.552,Z 766.457,A -85,B 0,C 180,E1 -5503.785,E2 -5503.785} C_VEL
LIN {X 0,Y 511.766,Z 753.482,A -85,B 0,C 180,E1 -5504.057,E2 -5504.057} C_VEL
LIN {X 0,Y 512.15,Z 659.554,A -85,B 0,C 180,E1 -5505.384,E2 -5505.384} C_VEL
LIN {X 0,Y 510.715,Z 648.208,A -85,B 0,C 180,E1 -5505.603,E2 -5505.603} C_VEL
LIN {X 0,Y 511.402,Z 619.55,A -85,B 0,C 180,E1 -5509.028,E2 -5509.028} C_VEL
LIN {X 0,Y 512.089,Z 595.173,A -85,B 0,C 180,E1 -5511.961,E2 -5511.961} C_VEL
LIN {X 0,Y 512.493,Z 579.637,A -85,B 0,C 180,E1 -5513.862,E2 -5513.862} C_VEL
LIN {X 0,Y 510.389,Z 569.16,A -85,B 0,C 180,E1 -5515.268,E2 -5515.268} C_VEL
LIN {X 0,Y 509.918,Z 566.971,A -85,B 0,C 180,E1 -5515.566,E2 -5515.566} C_VEL
LIN {X 0,Y 509.877,Z 566.97,A -85,B 0,C 180,E1 -5518.843,E2 -5518.843} C_VEL
LIN {X 0,Y 509.821,Z 566.98,A -85,B 0,C 180,E1 -5521.589,E2 -5521.589} C_VEL
LIN {X 0,Y 509.853,Z 566.974,A -85,B 0,C 180,E1 -5524.412,E2 -5524.412} C_VEL
LIN {X 0,Y 509.817,Z 566.976,A -85,B 0,C 180,E1 -5527.34,E2 -5527.34} C_VEL
LIN {X 0,Y 509.858,Z 566.974,A -85,B 0,C 180,E1 -5530.379,E2 -5530.379} C_VEL
LIN {X 0,Y 509.82,Z 566.974,A -85,B 0,C 180,E1 -5533.061,E2 -5533.061} C_VEL
LIN {X 0,Y 509.826,Z 566.977,A -85,B 0,C 180,E1 -5535.791,E2 -5535.791} C_VEL
LIN {X 0,Y 509.861,Z 566.972,A -85,B 0,C 180,E1 -5538.575,E2 -5538.575} C_VEL
LIN {X 0,Y 509.851,Z 566.972,A -85,B 0,C 180,E1 -5541.785,E2 -5541.785} C_VEL
LIN {X 0,Y 509.84,Z 566.971,A -85,B 0,C 180,E1 -5544.623,E2 -5544.623} C_VEL
LIN {X 0,Y 509.858,Z 566.969,A -85,B 0,C 180,E1 -5547.481,E2 -5547.481} C_VEL
LIN {X 0,Y 509.874,Z 566.972,A -85,B 0,C 180,E1 -5550.268,E2 -5550.268} C_VEL
LIN {X 0,Y 509.879,Z 566.969,A -85,B 0,C 180,E1 -5552.944,E2 -5552.944} C_VEL
LIN {X 0,Y 509.861,Z 566.969,A -85,B 0,C 180,E1 -5555.573,E2 -5555.573} C_VEL
LIN {X 0,Y 509.842,Z 566.973,A -85,B 0,C 180,E1 -5558.998,E2 -5558.998} C_VEL
LIN {X 0,Y 509.879,Z 566.969,A -85,B 0,C 180,E1 -5561.999,E2 -5561.999} C_VEL
LIN {X 0,Y 509.9,Z 566.967,A -85,B 0,C 180,E1 -5564.818,E2 -5564.818} C_VEL
LIN {X 0,Y 509.895,Z 566.968,A -85,B 0,C 180,E1 -5568.121,E2 -5568.121} C_VEL
LIN {X 0,Y 509.909,Z 566.958,A -85,B 0,C 180,E1 -5571.28,E2 -5571.28} C_VEL
LIN {X 0,Y 509.973,Z 566.955,A -85,B 0,C 180,E1 -5573.67,E2 -5573.67} C_VEL
LIN {X 0,Y 509.951,Z 566.96,A -85,B 0,C 180,E1 -5576.84,E2 -5576.84} C_VEL
LIN {X 0,Y 510.056,Z 566.944,A -85,B 0,C 180,E1 -5579.21,E2 -5579.21} C_VEL
LIN {X 0,Y 510.046,Z 566.95,A -85,B 0,C 180,E1 -5582.369,E2 -5582.369} C_VEL
LIN {X 0,Y 509.972,Z 566.951,A -85,B 0,C 180,E1 -5586.33,E2 -5586.33} C_VEL
LIN {X 0,Y 509.909,Z 566.97,A -85,B 0,C 180,E1 -5588.72,E2 -5588.72} C_VEL
LIN {X 0,Y 509.895,Z 566.96,A -85,B 0,C 180,E1 -5591.932,E2 -5591.932} C_VEL
LIN {X 0,Y 509.883,Z 566.971,A -85,B 0,C 180,E1 -5595.242,E2 -5595.242} C_VEL
LIN {X 0,Y 509.879,Z 566.964,A -85,B 0,C 180,E1 -5598.001,E2 -5598.001} C_VEL
LIN {X 0,Y 509.841,Z 566.979,A -85,B 0,C 180,E1 -5601.002,E2 -5601.002} C_VEL
LIN {X 0,Y 509.861,Z 566.968,A -85,B 0,C 180,E1 -5604.427,E2 -5604.427} C_VEL
LIN {X 0,Y 509.88,Z 566.976,A -85,B 0,C 180,E1 -5607.056,E2 -5607.056} C_VEL
LIN {X 0,Y 509.873,Z 566.966,A -85,B 0,C 180,E1 -5609.75,E2 -5609.75} C_VEL
LIN {X 0,Y 509.869,Z 566.973,A -85,B 0,C 180,E1 -5612.776,E2 -5612.776} C_VEL
LIN {X 0,Y 509.836,Z 566.976,A -85,B 0,C 180,E1 -5615.582,E2 -5615.582} C_VEL
LIN {X 0,Y 509.846,Z 566.971,A -85,B 0,C 180,E1 -5618.339,E2 -5618.339} C_VEL
LIN {X 0,Y 509.853,Z 566.966,A -85,B 0,C 180,E1 -5621.426,E2 -5621.426} C_VEL
LIN {X 0,Y 509.852,Z 566.972,A -85,B 0,C 180,E1 -5624.669,E2 -5624.669} C_VEL
LIN {X 0,Y 509.853,Z 566.968,A -85,B 0,C 180,E1 -5628.104,E2 -5628.104} C_VEL
LIN {X 0,Y 509.844,Z 566.973,A -85,B 0,C 180,E1 -5630.649,E2 -5630.649} C_VEL
LIN {X 0,Y 509.829,Z 566.978,A -85,B 0,C 180,E1 -5633.752,E2 -5633.752} C_VEL
LIN {X 0,Y 509.164,Z 567.058,A -85,B 0,C 180,E1 -5634.412,E2 -5634.412} C_VEL
LIN {X 0,Y 506.346,Z 567.415,A -85,B 0,C 180,E1 -5635.484,E2 -5635.484} C_VEL
LIN {X 0,Y 503.953,Z 567.712,A -85,B 0,C 180,E1 -5636.347,E2 -5636.347} C_VEL
LIN {X 0,Y 502.903,Z 567.84,A -85,B 0,C 180,E1 -5637.014,E2 -5637.014} C_VEL
LIN {X 0,Y 502.806,Z 567.851,A -85,B 0,C 180,E1 -5637.239,E2 -5637.239} C_VEL
LIN {X 0,Y 502.814,Z 567.851,A -85,B 0,C 180,E1 -5640.066,E2 -5640.066} C_VEL
LIN {X 0,Y 502.863,Z 567.98,A -85,B 0,C 180,E1 -5642.279,E2 -5642.279} C_VEL
LIN {X 0,Y 504.679,Z 574.151,A -85,B 0,C 180,E1 -5642.429,E2 -5642.429} C_VEL
LIN {X 0,Y 505.408,Z 577.774,A -85,B 0,C 180,E1 -5642.506,E2 -5642.506} C_VEL
LIN {X 0,Y 504.899,Z 672.738,A -85,B 0,C 180,E1 -5643.884,E2 -5643.884} C_VEL
LIN {X 0,Y 504.682,Z 685.937,A -85,B 0,C 180,E1 -5644.232,E2 -5644.232} C_VEL
LIN {X 0,Y 504.484,Z 698.271,A -85,B 0,C 180,E1 -5644.73,E2 -5644.73} C_VEL
LIN {X 0,Y 504.168,Z 710.412,A -85,B 0,C 180,E1 -5645.39,E2 -5645.39} C_VEL
LIN {X 0,Y 503.807,Z 721.139,A -85,B 0,C 180,E1 -5646.138,E2 -5646.138} C_VEL
LIN {X 0,Y 503.432,Z 730.933,A -85,B 0,C 180,E1 -5646.991,E2 -5646.991} C_VEL
LIN {X 0,Y 503.12,Z 740.833,A -85,B 0,C 180,E1 -5648.059,E2 -5648.059} C_VEL
LIN {X 0,Y 502.827,Z 748.862,A -85,B 0,C 180,E1 -5649.121,E2 -5649.121} C_VEL
LIN {X 0,Y 502.602,Z 756.584,A -85,B 0,C 180,E1 -5650.392,E2 -5650.392} C_VEL
LIN {X 0,Y 502.409,Z 762.873,A -85,B 0,C 180,E1 -5651.697,E2 -5651.697} C_VEL
LIN {X 0,Y 502.281,Z 767.447,A -85,B 0,C 180,E1 -5652.913,E2 -5652.913} C_VEL
LIN {X 0,Y 502.218,Z 769.955,A -85,B 0,C 180,E1 -5653.747,E2 -5653.747} C_VEL
LIN {X 0,Y 502.145,Z 772.728,A -85,B 0,C 180,E1 -5654.956,E2 -5654.956} C_VEL
LIN {X 0,Y 502.056,Z 774.636,A -85,B 0,C 180,E1 -5656.233,E2 -5656.233} C_VEL
LIN {X 0,Y 502.093,Z 775.603,A -85,B 0,C 180,E1 -5657.88,E2 -5657.88} C_VEL
LIN {X 0,Y 502.158,Z 775.49,A -85,B 0,C 180,E1 -5658.701,E2 -5658.701} C_VEL
LIN {X 0,Y 502.122,Z 774.947,A -85,B 0,C 180,E1 -5659.517,E2 -5659.517} C_VEL
LIN {X 0,Y 502.114,Z 772.697,A -85,B 0,C 180,E1 -5661.143,E2 -5661.143} C_VEL
LIN {X 0,Y 502.252,Z 769.879,A -85,B 0,C 180,E1 -5662.361,E2 -5662.361} C_VEL
LIN {X 0,Y 502.338,Z 766.062,A -85,B 0,C 180,E1 -5663.574,E2 -5663.574} C_VEL
LIN {X 0,Y 502.403,Z 761.142,A -85,B 0,C 180,E1 -5664.783,E2 -5664.783} C_VEL
LIN {X 0,Y 502.623,Z 754.921,A -85,B 0,C 180,E1 -5665.991,E2 -5665.991} C_VEL
LIN {X 0,Y 502.824,Z 747.216,A -85,B 0,C 180,E1 -5667.196,E2 -5667.196} C_VEL
LIN {X 0,Y 503.136,Z 739.35,A -85,B 0,C 180,E1 -5668.199,E2 -5668.199} C_VEL
LIN {X 0,Y 503.473,Z 729.806,A -85,B 0,C 180,E1 -5669.2,E2 -5669.2} C_VEL
LIN {X 0,Y 503.748,Z 719.133,A -85,B 0,C 180,E1 -5670.1,E2 -5670.1} C_VEL
LIN {X 0,Y 504.243,Z 707.063,A -85,B 0,C 180,E1 -5670.898,E2 -5670.898} C_VEL
LIN {X 0,Y 504.507,Z 695.193,A -85,B 0,C 180,E1 -5671.497,E2 -5671.497} C_VEL
LIN {X 0,Y 504.761,Z 682.212,A -85,B 0,C 180,E1 -5671.97,E2 -5671.97} C_VEL
LIN {X 0,Y 504.96,Z 669.418,A -85,B 0,C 180,E1 -5672.268,E2 -5672.268} C_VEL
LIN {X 0,Y 505.351,Z 575.856,A -85,B 0,C 180,E1 -5673.613,E2 -5673.613} C_VEL
LIN {X 0,Y 502.804,Z 567.857,A -85,B 0,C 180,E1 -5673.832,E2 -5673.832} C_VEL
LIN {X 0,Y 502.909,Z 567.841,A -85,B 0,C 180,E1 -5676.419,E2 -5676.419} C_VEL
LIN {X 0,Y 502.867,Z 567.842,A -85,B 0,C 180,E1 -5678.843,E2 -5678.843} C_VEL
LIN {X 0,Y 502.896,Z 567.846,A -85,B 0,C 180,E1 -5682.1,E2 -5682.1} C_VEL
LIN {X 0,Y 502.851,Z 567.844,A -85,B 0,C 180,E1 -5685.399,E2 -5685.399} C_VEL
LIN {X 0,Y 502.848,Z 567.852,A -85,B 0,C 180,E1 -5688.122,E2 -5688.122} C_VEL
LIN {X 0,Y 502.83,Z 567.847,A -85,B 0,C 180,E1 -5690.536,E2 -5690.536} C_VEL
LIN {X 0,Y 502.79,Z 567.85,A -85,B 0,C 180,E1 -5693.04,E2 -5693.04} C_VEL
LIN {X 0,Y 502.822,Z 567.851,A -85,B 0,C 180,E1 -5695.676,E2 -5695.676} C_VEL
LIN {X 0,Y 502.841,Z 567.851,A -85,B 0,C 180,E1 -5698.372,E2 -5698.372} C_VEL
LIN {X 0,Y 502.883,Z 567.909,A -85,B 0,C 180,E1 -5700.28,E2 -5700.28} C_VEL
LIN {X 0,Y 505.178,Z 575.44,A -85,B 0,C 180,E1 -5700.468,E2 -5700.468} C_VEL
LIN {X 0,Y 505.52,Z 578.425,A -85,B 0,C 180,E1 -5700.524,E2 -5700.524} C_VEL
LIN {X 0,Y 504.864,Z 672.663,A -85,B 0,C 180,E1 -5701.9,E2 -5701.9} C_VEL
LIN {X 0,Y 504.687,Z 685.575,A -85,B 0,C 180,E1 -5702.243,E2 -5702.243} C_VEL
LIN {X 0,Y 504.412,Z 699.203,A -85,B 0,C 180,E1 -5702.795,E2 -5702.795} C_VEL
LIN {X 0,Y 504.129,Z 710.572,A -85,B 0,C 180,E1 -5703.427,E2 -5703.427} C_VEL
LIN {X 0,Y 503.766,Z 720.748,A -85,B 0,C 180,E1 -5704.138,E2 -5704.138} C_VEL
LIN {X 0,Y 503.494,Z 729.757,A -85,B 0,C 180,E1 -5704.909,E2 -5704.909} C_VEL
LIN {X 0,Y 503.142,Z 739.453,A -85,B 0,C 180,E1 -5705.92,E2 -5705.92} C_VEL
LIN {X 0,Y 502.813,Z 749.122,A -85,B 0,C 180,E1 -5707.183,E2 -5707.183} C_VEL
LIN {X 0,Y 502.575,Z 755.484,A -85,B 0,C 180,E1 -5708.21,E2 -5708.21} C_VEL
LIN {X 0,Y 502.45,Z 761.268,A -85,B 0,C 180,E1 -5709.352,E2 -5709.352} C_VEL
LIN {X 0,Y 502.296,Z 765.912,A -85,B 0,C 180,E1 -5710.489,E2 -5710.489} C_VEL
LIN {X 0,Y 502.219,Z 769.544,A -85,B 0,C 180,E1 -5711.62,E2 -5711.62} C_VEL
LIN {X 0,Y 502.126,Z 772.289,A -85,B 0,C 180,E1 -5712.746,E2 -5712.746} C_VEL
LIN {X 0,Y 502.07,Z 774.842,A -85,B 0,C 180,E1 -5714.447,E2 -5714.447} C_VEL
LIN {X 0,Y 502.035,Z 775.554,A -85,B 0,C 180,E1 -5715.577,E2 -5715.577} C_VEL
LIN {X 0,Y 502.024,Z 775.493,A -85,B 0,C 180,E1 -5716.714,E2 -5716.714} C_VEL
LIN {X 0,Y 502.07,Z 774.602,A -85,B 0,C 180,E1 -5717.892,E2 -5717.892} C_VEL
LIN {X 0,Y 502.108,Z 772.804,A -85,B 0,C 180,E1 -5719.097,E2 -5719.097} C_VEL
LIN {X 0,Y 502.179,Z 769.999,A -85,B 0,C 180,E1 -5720.328,E2 -5720.328} C_VEL
LIN {X 0,Y 502.304,Z 766.062,A -85,B 0,C 180,E1 -5721.583,E2 -5721.583} C_VEL
LIN {X 0,Y 502.45,Z 760.077,A -85,B 0,C 180,E1 -5723.025,E2 -5723.025} C_VEL
LIN {X 0,Y 502.719,Z 752.524,A -85,B 0,C 180,E1 -5724.403,E2 -5724.403} C_VEL
LIN {X 0,Y 502.954,Z 744.798,A -85,B 0,C 180,E1 -5725.529,E2 -5725.529} C_VEL
LIN {X 0,Y 503.263,Z 736.643,A -85,B 0,C 180,E1 -5726.506,E2 -5726.506} C_VEL
LIN {X 0,Y 503.6,Z 726.491,A -85,B 0,C 180,E1 -5727.501,E2 -5727.501} C_VEL
LIN {X 0,Y 504.008,Z 715.279,A -85,B 0,C 180,E1 -5728.374,E2 -5728.374} C_VEL
LIN {X 0,Y 504.294,Z 703.966,A -85,B 0,C 180,E1 -5729.063,E2 -5729.063} C_VEL
LIN {X 0,Y 504.557,Z 692.577,A -85,B 0,C 180,E1 -5729.596,E2 -5729.596} C_VEL
LIN {X 0,Y 504.718,Z 680.249,A -85,B 0,C 180,E1 -5730.016,E2 -5730.016} C_VEL
LIN {X 0,Y 504.95,Z 666.359,A -85,B 0,C 180,E1 -5730.304,E2 -5730.304} C_VEL
LIN {X 0,Y 505.325,Z 577.532,A -85,B 0,C 180,E1 -5731.593,E2 -5731.593} C_VEL
LIN {X 0,Y 503.915,Z 571.384,A -85,B 0,C 180,E1 -5731.731,E2 -5731.731} C_VEL
LIN {X 0,Y 502.852,Z 567.85,A -85,B 0,C 180,E1 -5731.837,E2 -5731.837} C_VEL
LIN {X 0,Y 502.833,Z 567.852,A -85,B 0,C 180,E1 -5734.324,E2 -5734.324} C_VEL
LIN {X 0,Y 502.801,Z 567.852,A -85,B 0,C 180,E1 -5737.295,E2 -5737.295} C_VEL
LIN {X 0,Y 502.817,Z 567.855,A -85,B 0,C 180,E1 -5740.4,E2 -5740.4} C_VEL
LIN {X 0,Y 502.827,Z 567.851,A -85,B 0,C 180,E1 -5742.931,E2 -5742.931} C_VEL
LIN {X 0,Y 502.835,Z 567.846,A -85,B 0,C 180,E1 -5745.429,E2 -5745.429} C_VEL
LIN {X 0,Y 502.885,Z 567.846,A -85,B 0,C 180,E1 -5748.717,E2 -5748.717} C_VEL
LIN {X 0,Y 502.892,Z 567.84,A -85,B 0,C 180,E1 -5751.967,E2 -5751.967} C_VEL
LIN {X 0,Y 502.95,Z 567.838,A -85,B 0,C 180,E1 -5754.387,E2 -5754.387} C_VEL
LIN {X 0,Y 503.016,Z 567.821,A -85,B 0,C 180,E1 -5757.598,E2 -5757.598} C_VEL
LIN {X 0,Y 503.016,Z 567.825,A -85,B 0,C 180,E1 -5760,E2 -5760} C_VEL
LIN {X 0,Y 503.015,Z 567.83,A -85,B 0,C 180,E1 -5762.402,E2 -5762.402} C_VEL
LIN {X 0,Y 502.953,Z 567.83,A -85,B 0,C 180,E1 -5765.613,E2 -5765.613} C_VEL
LIN {X 0,Y 502.892,Z 567.838,A -85,B 0,C 180,E1 -5768.034,E2 -5768.034} C_VEL
LIN {X 0,Y 502.885,Z 567.837,A -85,B 0,C 180,E1 -5771.283,E2 -5771.283} C_VEL
LIN {X 0,Y 502.842,Z 567.849,A -85,B 0,C 180,E1 -5774.571,E2 -5774.571} C_VEL
LIN {X 0,Y 502.852,Z 567.841,A -85,B 0,C 180,E1 -5777.907,E2 -5777.907} C_VEL
LIN {X 0,Y 502.821,Z 567.851,A -85,B 0,C 180,E1 -5780.537,E2 -5780.537} C_VEL
LIN {X 0,Y 502.797,Z 567.85,A -85,B 0,C 180,E1 -5783.04,E2 -5783.04} C_VEL
LIN {X 0,Y 502.834,Z 567.846,A -85,B 0,C 180,E1 -5785.676,E2 -5785.676} C_VEL
LIN {X 0,Y 502.835,Z 567.85,A -85,B 0,C 180,E1 -5788.373,E2 -5788.373} C_VEL
LIN {X 0,Y 502.79,Z 567.85,A -85,B 0,C 180,E1 -5791.5,E2 -5791.5} C_VEL
LIN {X 0,Y 502.8,Z 567.855,A -85,B 0,C 180,E1 -5794.446,E2 -5794.446} C_VEL
LIN {X 0,Y 502.776,Z 567.854,A -85,B 0,C 180,E1 -5797.179,E2 -5797.179} C_VEL
LIN {X 0,Y 502.821,Z 567.849,A -85,B 0,C 180,E1 -5800.012,E2 -5800.012} C_VEL
LIN {X 0,Y 502.825,Z 567.85,A -85,B 0,C 180,E1 -5802.203,E2 -5802.203} C_VEL
LIN {X 0,Y 502.796,Z 567.851,A -85,B 0,C 180,E1 -5805.469,E2 -5805.469} C_VEL
LIN {X 0,Y 502.817,Z 567.851,A -85,B 0,C 180,E1 -5808.935,E2 -5808.935} C_VEL
LIN {X 0,Y 502.791,Z 567.855,A -85,B 0,C 180,E1 -5812.047,E2 -5812.047} C_VEL
LIN {X 0,Y 502.802,Z 567.853,A -85,B 0,C 180,E1 -5815.035,E2 -5815.035} C_VEL
LIN {X 0,Y 502.784,Z 567.856,A -85,B 0,C 180,E1 -5817.916,E2 -5817.916} C_VEL
LIN {X 0,Y 502.823,Z 567.854,A -85,B 0,C 180,E1 -5820.713,E2 -5820.713} C_VEL
LIN {X 0,Y 502.861,Z 567.893,A -85,B 0,C 180,E1 -5822.804,E2 -5822.804} C_VEL
LIN {X 0,Y 505.241,Z 580.274,A -85,B 0,C 180,E1 -5824.711,E2 -5824.711} C_VEL
LIN {X 0,Y 504.693,Z 598.277,A -85,B 0,C 180,E1 -5827.268,E2 -5827.268} C_VEL
LIN {X 0,Y 504.173,Z 619.567,A -85,B 0,C 180,E1 -5830.243,E2 -5830.243} C_VEL
LIN {X 0,Y 503.496,Z 645.275,A -85,B 0,C 180,E1 -5833.79,E2 -5833.79} C_VEL
LIN {X 0,Y 503.456,Z 648.09,A -85,B 0,C 180,E1 -5834.177,E2 -5834.177} C_VEL
LIN {X 0,Y 505.346,Z 662.961,A -85,B 0,C 180,E1 -5834.467,E2 -5834.467} C_VEL
LIN {X 0,Y 504.807,Z 757.942,A -85,B 0,C 180,E1 -5835.848,E2 -5835.848} C_VEL
LIN {X 0,Y 504.483,Z 771.18,A -85,B 0,C 180,E1 -5836.198,E2 -5836.198} C_VEL
LIN {X 0,Y 504.22,Z 783.96,A -85,B 0,C 180,E1 -5836.704,E2 -5836.704} C_VEL
LIN {X 0,Y 503.857,Z 796.04,A -85,B 0,C 180,E1 -5837.354,E2 -5837.354} C_VEL
LIN {X 0,Y 503.49,Z 808.414,A -85,B 0,C 180,E1 -5838.221,E2 -5838.221} C_VEL
LIN {X 0,Y 503.129,Z 818.772,A -85,B 0,C 180,E1 -5839.131,E2 -5839.131} C_VEL
LIN {X 0,Y 502.835,Z 828.09,A -85,B 0,C 180,E1 -5840.142,E2 -5840.142} C_VEL
LIN {X 0,Y 502.569,Z 837.167,A -85,B 0,C 180,E1 -5841.354,E2 -5841.354} C_VEL
LIN {X 0,Y 502.355,Z 844.486,A -85,B 0,C 180,E1 -5842.565,E2 -5842.565} C_VEL
LIN {X 0,Y 502.235,Z 849.42,A -85,B 0,C 180,E1 -5843.573,E2 -5843.573} C_VEL
LIN {X 0,Y 502.186,Z 854.228,A -85,B 0,C 180,E1 -5844.781,E2 -5844.781} C_VEL
LIN {X 0,Y 502.2,Z 857.91,A -85,B 0,C 180,E1 -5845.988,E2 -5845.988} C_VEL
LIN {X 0,Y 502.122,Z 859.804,A -85,B 0,C 180,E1 -5846.791,E2 -5846.791} C_VEL
LIN {X 0,Y 502.12,Z 861.227,A -85,B 0,C 180,E1 -5847.594,E2 -5847.594} C_VEL
LIN {X 0,Y 502,Z 862.85,A -85,B 0,C 180,E1 -5849.198,E2 -5849.198} C_VEL
LIN {X 0,Y 501.993,Z 863.074,A -85,B 0,C 180,E1 -5850,E2 -5850} C_VEL
LIN {X 0,Y 502,Z 862.857,A -85,B 0,C 180,E1 -5850.802,E2 -5850.802} C_VEL
LIN {X 0,Y 502.12,Z 861.242,A -85,B 0,C 180,E1 -5852.406,E2 -5852.406} C_VEL
LIN {X 0,Y 502.122,Z 859.827,A -85,B 0,C 180,E1 -5853.209,E2 -5853.209} C_VEL
LIN {X 0,Y 502.15,Z 856.854,A -85,B 0,C 180,E1 -5854.415,E2 -5854.415} C_VEL
LIN {X 0,Y 502.255,Z 852.833,A -85,B 0,C 180,E1 -5855.621,E2 -5855.621} C_VEL
LIN {X 0,Y 502.333,Z 846.736,A -85,B 0,C 180,E1 -5857.011,E2 -5857.011} C_VEL
LIN {X 0,Y 502.504,Z 839.87,A -85,B 0,C 180,E1 -5858.242,E2 -5858.242} C_VEL
LIN {X 0,Y 502.741,Z 831.486,A -85,B 0,C 180,E1 -5859.454,E2 -5859.454} C_VEL
LIN {X 0,Y 503.01,Z 822.888,A -85,B 0,C 180,E1 -5860.465,E2 -5860.465} C_VEL
LIN {X 0,Y 503.397,Z 812.281,A -85,B 0,C 180,E1 -5861.475,E2 -5861.475} C_VEL
LIN {X 0,Y 503.688,Z 800.334,A -85,B 0,C 180,E1 -5862.388,E2 -5862.388} C_VEL
LIN {X 0,Y 504.098,Z 788.316,A -85,B 0,C 180,E1 -5863.094,E2 -5863.094} C_VEL
LIN {X 0,Y 504.44,Z 775.817,A -85,B 0,C 180,E1 -5863.649,E2 -5863.649} C_VEL
LIN {X 0,Y 504.723,Z 762.883,A -85,B 0,C 180,E1 -5864.052,E2 -5864.052} C_VEL
LIN {X 0,Y 504.923,Z 747.404,A -85,B 0,C 180,E1 -5864.329,E2 -5864.329} C_VEL
LIN {X 0,Y 505.338,Z 660.617,A -85,B 0,C 180,E1 -5865.573,E2 -5865.573} C_VEL
LIN {X 0,Y 503.71,Z 647.656,A -85,B 0,C 180,E1 -5865.823,E2 -5865.823} C_VEL
LIN {X 0,Y 504.433,Z 620.573,A -85,B 0,C 180,E1 -5869.111,E2 -5869.111} C_VEL
LIN {X 0,Y 505.179,Z 594.643,A -85,B 0,C 180,E1 -5872.277,E2 -5872.277} C_VEL
LIN {X 0,Y 505.595,Z 580.878,A -85,B 0,C 180,E1 -5873.99,E2 -5873.99} C_VEL
LIN {X 0,Y 502.888,Z 567.846,A -85,B 0,C 180,E1 -5875.783,E2 -5875.783} C_VEL
LIN {X 0,Y 502.841,Z 567.849,A -85,B 0,C 180,E1 -5878.372,E2 -5878.372} C_VEL
LIN {X 0,Y 502.793,Z 567.855,A -85,B 0,C 180,E1 -5881.498,E2 -5881.498} C_VEL
LIN {X 0,Y 502.806,Z 567.852,A -85,B 0,C 180,E1 -5884.444,E2 -5884.444} C_VEL
LIN {X 0,Y 502.779,Z 567.852,A -85,B 0,C 180,E1 -5887.178,E2 -5887.178} C_VEL
LIN {X 0,Y 502.819,Z 567.855,A -85,B 0,C 180,E1 -5890.011,E2 -5890.011} C_VEL
LIN {X 0,Y 502.769,Z 567.853,A -85,B 0,C 180,E1 -5893.23,E2 -5893.23} C_VEL
LIN {X 0,Y 502.785,Z 567.852,A -85,B 0,C 180,E1 -5895.66,E2 -5895.66} C_VEL
LIN {X 0,Y 502.825,Z 567.85,A -85,B 0,C 180,E1 -5897.863,E2 -5897.863} C_VEL
LIN {X 0,Y 502.816,Z 567.845,A -85,B 0,C 180,E1 -5901.025,E2 -5901.025} C_VEL
LIN {X 0,Y 502.78,Z 567.858,A -85,B 0,C 180,E1 -5904.166,E2 -5904.166} C_VEL
LIN {X 0,Y 502.826,Z 567.846,A -85,B 0,C 180,E1 -5906.992,E2 -5906.992} C_VEL
LIN {X 0,Y 502.823,Z 567.85,A -85,B 0,C 180,E1 -5910.061,E2 -5910.061} C_VEL
LIN {X 0,Y 502.827,Z 567.852,A -85,B 0,C 180,E1 -5912.533,E2 -5912.533} C_VEL
LIN {X 0,Y 502.82,Z 567.846,A -85,B 0,C 180,E1 -5915.298,E2 -5915.298} C_VEL
LIN {X 0,Y 502.772,Z 567.847,A -85,B 0,C 180,E1 -5917.826,E2 -5917.826} C_VEL
LIN {X 0,Y 502.817,Z 567.855,A -85,B 0,C 180,E1 -5920.4,E2 -5920.4} C_VEL
LIN {X 0,Y 502.826,Z 567.843,A -85,B 0,C 180,E1 -5922.931,E2 -5922.931} C_VEL
LIN {X 0,Y 502.835,Z 567.842,A -85,B 0,C 180,E1 -5925.429,E2 -5925.429} C_VEL
LIN {X 0,Y 502.871,Z 567.844,A -85,B 0,C 180,E1 -5928.717,E2 -5928.717} C_VEL
LIN {X 0,Y 502.892,Z 567.832,A -85,B 0,C 180,E1 -5931.966,E2 -5931.966} C_VEL
LIN {X 0,Y 502.953,Z 567.834,A -85,B 0,C 180,E1 -5934.387,E2 -5934.387} C_VEL
LIN {X 0,Y 503.016,Z 567.817,A -85,B 0,C 180,E1 -5937.598,E2 -5937.598} C_VEL
LIN {X 0,Y 503.016,Z 567.819,A -85,B 0,C 180,E1 -5940,E2 -5940} C_VEL
LIN {X 0,Y 503.015,Z 567.826,A -85,B 0,C 180,E1 -5942.402,E2 -5942.402} C_VEL
LIN {X 0,Y 502.941,Z 567.824,A -85,B 0,C 180,E1 -5945.613,E2 -5945.613} C_VEL
LIN {X 0,Y 502.892,Z 567.837,A -85,B 0,C 180,E1 -5948.033,E2 -5948.033} C_VEL
LIN {X 0,Y 502.872,Z 567.838,A -85,B 0,C 180,E1 -5951.283,E2 -5951.283} C_VEL
LIN {X 0,Y 502.835,Z 567.847,A -85,B 0,C 180,E1 -5954.571,E2 -5954.571} C_VEL
LIN {X 0,Y 502.852,Z 567.839,A -85,B 0,C 180,E1 -5957.907,E2 -5957.907} C_VEL
LIN {X 0,Y 502.819,Z 567.847,A -85,B 0,C 180,E1 -5960.537,E2 -5960.537} C_VEL
LIN {X 0,Y 502.785,Z 567.857,A -85,B 0,C 180,E1 -5963.041,E2 -5963.041} C_VEL
LIN {X 0,Y 502.833,Z 567.845,A -85,B 0,C 180,E1 -5965.676,E2 -5965.676} C_VEL
LIN {X 0,Y 502.835,Z 567.845,A -85,B 0,C 180,E1 -5968.373,E2 -5968.373} C_VEL
LIN {X 0,Y 502.79,Z 567.854,A -85,B 0,C 180,E1 -5971.5,E2 -5971.5} C_VEL
LIN {X 0,Y 502.799,Z 567.847,A -85,B 0,C 180,E1 -5974.445,E2 -5974.445} C_VEL
LIN {X 0,Y 502.777,Z 567.86,A -85,B 0,C 180,E1 -5977.18,E2 -5977.18} C_VEL
LIN {X 0,Y 502.783,Z 567.85,A -85,B 0,C 180,E1 -5980.016,E2 -5980.016} C_VEL
LIN {X 0,Y 502.798,Z 567.839,A -85,B 0,C 180,E1 -5982.2,E2 -5982.2} C_VEL
LIN {X 0,Y 502.796,Z 567.856,A -85,B 0,C 180,E1 -5985.469,E2 -5985.469} C_VEL
LIN {X 0,Y 502.817,Z 567.847,A -85,B 0,C 180,E1 -5988.935,E2 -5988.935} C_VEL
LIN {X 0,Y 502.791,Z 567.849,A -85,B 0,C 180,E1 -5992.047,E2 -5992.047} C_VEL
LIN {X 0,Y 502.808,Z 567.852,A -85,B 0,C 180,E1 -5995.036,E2 -5995.036} C_VEL
LIN {X 0,Y 502.806,Z 567.851,A -85,B 0,C 180,E1 -5997.239,E2 -5997.239} C_VEL
LIN {X 0,Y 502.105,Z 567.94,A -85,B 0,C 180,E1 -5997.908,E2 -5997.908} C_VEL
LIN {X 0,Y 499.24,Z 568.296,A -85,B 0,C 180,E1 -5998.994,E2 -5998.994} C_VEL
LIN {X 0,Y 496.846,Z 568.596,A -85,B 0,C 180,E1 -5999.869,E2 -5999.869} C_VEL
LIN {X 0,Y 495.83,Z 568.72,A -85,B 0,C 180,E1 -6000.544,E2 -6000.544} C_VEL
LIN {X 0,Y 495.753,Z 568.73,A -85,B 0,C 180,E1 -6000.773,E2 -6000.773} C_VEL
LIN {X 0,Y 495.827,Z 568.725,A -85,B 0,C 180,E1 -6002.048,E2 -6002.048} C_VEL
LIN {X 0,Y 498.037,Z 576.001,A -85,B 0,C 180,E1 -6002.236,E2 -6002.236} C_VEL
LIN {X 0,Y 498.636,Z 580.553,A -85,B 0,C 180,E1 -6002.323,E2 -6002.323} C_VEL
LIN {X 0,Y 498.044,Z 673.693,A -85,B 0,C 180,E1 -6003.694,E2 -6003.694} C_VEL
LIN {X 0,Y 497.828,Z 686.77,A -85,B 0,C 180,E1 -6004.047,E2 -6004.047} C_VEL
LIN {X 0,Y 497.624,Z 698.568,A -85,B 0,C 180,E1 -6004.529,E2 -6004.529} C_VEL
LIN {X 0,Y 497.307,Z 709.816,A -85,B 0,C 180,E1 -6005.139,E2 -6005.139} C_VEL
LIN {X 0,Y 496.931,Z 720.783,A -85,B 0,C 180,E1 -6005.898,E2 -6005.898} C_VEL
LIN {X 0,Y 496.533,Z 730.751,A -85,B 0,C 180,E1 -6006.758,E2 -6006.758} C_VEL
LIN {X 0,Y 496.2,Z 739.931,A -85,B 0,C 180,E1 -6007.736,E2 -6007.736} C_VEL
LIN {X 0,Y 495.897,Z 748.213,A -85,B 0,C 180,E1 -6008.815,E2 -6008.815} C_VEL
LIN {X 0,Y 495.582,Z 756.238,A -85,B 0,C 180,E1 -6010.102,E2 -6010.102} C_VEL
LIN {X 0,Y 495.432,Z 762.538,A -85,B 0,C 180,E1 -6011.387,E2 -6011.387} C_VEL
LIN {X 0,Y 495.265,Z 767.459,A -85,B 0,C 180,E1 -6012.663,E2 -6012.663} C_VEL
LIN {X 0,Y 495.158,Z 771.177,A -85,B 0,C 180,E1 -6013.933,E2 -6013.933} C_VEL
LIN {X 0,Y 495.059,Z 773.818,A -85,B 0,C 180,E1 -6015.195,E2 -6015.195} C_VEL
LIN {X 0,Y 494.999,Z 775.042,A -85,B 0,C 180,E1 -6016.033,E2 -6016.033} C_VEL
LIN {X 0,Y 494.985,Z 775.821,A -85,B 0,C 180,E1 -6016.87,E2 -6016.87} C_VEL
LIN {X 0,Y 495.049,Z 776.166,A -85,B 0,C 180,E1 -6018.397,E2 -6018.397} C_VEL
LIN {X 0,Y 495.073,Z 775.707,A -85,B 0,C 180,E1 -6019.366,E2 -6019.366} C_VEL
LIN {X 0,Y 495.034,Z 773.592,A -85,B 0,C 180,E1 -6021.016,E2 -6021.016} C_VEL
LIN {X 0,Y 495.182,Z 770.907,A -85,B 0,C 180,E1 -6022.251,E2 -6022.251} C_VEL
LIN {X 0,Y 495.292,Z 767.229,A -85,B 0,C 180,E1 -6023.482,E2 -6023.482} C_VEL
LIN {X 0,Y 495.363,Z 762.47,A -85,B 0,C 180,E1 -6024.709,E2 -6024.709} C_VEL
LIN {X 0,Y 495.573,Z 756.471,A -85,B 0,C 180,E1 -6025.934,E2 -6025.934} C_VEL
LIN {X 0,Y 495.796,Z 748.985,A -85,B 0,C 180,E1 -6027.156,E2 -6027.156} C_VEL
LIN {X 0,Y 496.184,Z 739.649,A -85,B 0,C 180,E1 -6028.377,E2 -6028.377} C_VEL
LIN {X 0,Y 496.551,Z 730.016,A -85,B 0,C 180,E1 -6029.392,E2 -6029.392} C_VEL
LIN {X 0,Y 496.862,Z 719.251,A -85,B 0,C 180,E1 -6030.304,E2 -6030.304} C_VEL
LIN {X 0,Y 497.319,Z 708.721,A -85,B 0,C 180,E1 -6031.012,E2 -6031.012} C_VEL
LIN {X 0,Y 497.644,Z 696.119,A -85,B 0,C 180,E1 -6031.669,E2 -6031.669} C_VEL
LIN {X 0,Y 497.889,Z 683.277,A -85,B 0,C 180,E1 -6032.149,E2 -6032.149} C_VEL
LIN {X 0,Y 498.108,Z 670.836,A -85,B 0,C 180,E1 -6032.451,E2 -6032.451} C_VEL
LIN {X 0,Y 498.539,Z 576.835,A -85,B 0,C 180,E1 -6033.824,E2 -6033.824} C_VEL
LIN {X 0,Y 495.749,Z 568.736,A -85,B 0,C 180,E1 -6034.039,E2 -6034.039} C_VEL
LIN {X 0,Y 495.863,Z 568.718,A -85,B 0,C 180,E1 -6036.51,E2 -6036.51} C_VEL
LIN {X 0,Y 495.837,Z 568.718,A -85,B 0,C 180,E1 -6038.97,E2 -6038.97} C_VEL
LIN {X 0,Y 495.855,Z 568.72,A -85,B 0,C 180,E1 -6042.275,E2 -6042.275} C_VEL
LIN {X 0,Y 495.81,Z 568.723,A -85,B 0,C 180,E1 -6045.623,E2 -6045.623} C_VEL
LIN {X 0,Y 495.808,Z 568.726,A -85,B 0,C 180,E1 -6048.247,E2 -6048.247} C_VEL
LIN {X 0,Y 495.775,Z 568.724,A -85,B 0,C 180,E1 -6050.756,E2 -6050.756} C_VEL
LIN {X 0,Y 495.743,Z 568.729,A -85,B 0,C 180,E1 -6053.387,E2 -6053.387} C_VEL
LIN {X 0,Y 495.824,Z 568.721,A -85,B 0,C 180,E1 -6056.749,E2 -6056.749} C_VEL
LIN {X 0,Y 495.828,Z 568.727,A -85,B 0,C 180,E1 -6060.038,E2 -6060.038} C_VEL
LIN {X 0,Y 498.516,Z 577.229,A -85,B 0,C 180,E1 -6060.274,E2 -6060.274} C_VEL
LIN {X 0,Y 498.579,Z 587.947,A -85,B 0,C 180,E1 -6060.438,E2 -6060.438} C_VEL
LIN {X 0,Y 497.992,Z 673.046,A -85,B 0,C 180,E1 -6061.701,E2 -6061.701} C_VEL
LIN {X 0,Y 497.797,Z 686.437,A -85,B 0,C 180,E1 -6062.064,E2 -6062.064} C_VEL
LIN {X 0,Y 497.533,Z 699.197,A -85,B 0,C 180,E1 -6062.584,E2 -6062.584} C_VEL
LIN {X 0,Y 497.232,Z 710.463,A -85,B 0,C 180,E1 -6063.209,E2 -6063.209} C_VEL
LIN {X 0,Y 496.85,Z 721.236,A -85,B 0,C 180,E1 -6063.967,E2 -6063.967} C_VEL
LIN {X 0,Y 496.535,Z 731.022,A -85,B 0,C 180,E1 -6064.821,E2 -6064.821} C_VEL
LIN {X 0,Y 496.167,Z 739.564,A -85,B 0,C 180,E1 -6065.725,E2 -6065.725} C_VEL
LIN {X 0,Y 495.913,Z 747.567,A -85,B 0,C 180,E1 -6066.751,E2 -6066.751} C_VEL
LIN {X 0,Y 495.557,Z 756.013,A -85,B 0,C 180,E1 -6068.09,E2 -6068.09} C_VEL
LIN {X 0,Y 495.406,Z 762.558,A -85,B 0,C 180,E1 -6069.418,E2 -6069.418} C_VEL
LIN {X 0,Y 495.242,Z 767.677,A -85,B 0,C 180,E1 -6070.751,E2 -6070.751} C_VEL
LIN {X 0,Y 495.161,Z 770.89,A -85,B 0,C 180,E1 -6071.841,E2 -6071.841} C_VEL
LIN {X 0,Y 495.061,Z 773.368,A -85,B 0,C 180,E1 -6072.953,E2 -6072.953} C_VEL
LIN {X 0,Y 495.021,Z 775.087,A -85,B 0,C 180,E1 -6074.079,E2 -6074.079} C_VEL
LIN {X 0,Y 494.962,Z 776.059,A -85,B 0,C 180,E1 -6075.23,E2 -6075.23} C_VEL
LIN {X 0,Y 494.949,Z 776.236,A -85,B 0,C 180,E1 -6076.398,E2 -6076.398} C_VEL
LIN {X 0,Y 495.007,Z 775.58,A -85,B 0,C 180,E1 -6077.584,E2 -6077.584} C_VEL
LIN {X 0,Y 495.064,Z 773.272,A -85,B 0,C 180,E1 -6079.23,E2 -6079.23} C_VEL
LIN {X 0,Y 495.115,Z 770.86,A -85,B 0,C 180,E1 -6080.3,E2 -6080.3} C_VEL
LIN {X 0,Y 495.26,Z 767.706,A -85,B 0,C 180,E1 -6081.363,E2 -6081.363} C_VEL
LIN {X 0,Y 495.401,Z 763.003,A -85,B 0,C 180,E1 -6082.601,E2 -6082.601} C_VEL
LIN {X 0,Y 495.582,Z 756.55,A -85,B 0,C 180,E1 -6083.932,E2 -6083.932} C_VEL
LIN {X 0,Y 495.849,Z 749.218,A -85,B 0,C 180,E1 -6085.135,E2 -6085.135} C_VEL
LIN {X 0,Y 496.253,Z 739.896,A -85,B 0,C 180,E1 -6086.352,E2 -6086.352} C_VEL
LIN {X 0,Y 496.558,Z 730.518,A -85,B 0,C 180,E1 -6087.344,E2 -6087.344} C_VEL
LIN {X 0,Y 496.962,Z 719.771,A -85,B 0,C 180,E1 -6088.261,E2 -6088.261} C_VEL
LIN {X 0,Y 497.314,Z 707.733,A -85,B 0,C 180,E1 -6089.066,E2 -6089.066} C_VEL
LIN {X 0,Y 497.64,Z 695.773,A -85,B 0,C 180,E1 -6089.676,E2 -6089.676} C_VEL
LIN {X 0,Y 497.86,Z 682.552,A -85,B 0,C 180,E1 -6090.158,E2 -6090.158} C_VEL
LIN {X 0,Y 498.003,Z 670.195,A -85,B 0,C 180,E1 -6090.447,E2 -6090.447} C_VEL
LIN {X 0,Y 498.557,Z 578.669,A -85,B 0,C 180,E1 -6091.802,E2 -6091.802} C_VEL
LIN {X 0,Y 497.197,Z 573.084,A -85,B 0,C 180,E1 -6091.933,E2 -6091.933} C_VEL
LIN {X 0,Y 495.848,Z 568.724,A -85,B 0,C 180,E1 -6092.065,E2 -6092.065} C_VEL
LIN {X 0,Y 495.771,Z 568.729,A -85,B 0,C 180,E1 -6095.126,E2 -6095.126} C_VEL
LIN {X 0,Y 495.735,Z 568.736,A -85,B 0,C 180,E1 -6098.371,E2 -6098.371} C_VEL
LIN {X 0,Y 495.776,Z 568.729,A -85,B 0,C 180,E1 -6100.971,E2 -6100.971} C_VEL
LIN {X 0,Y 495.771,Z 568.726,A -85,B 0,C 180,E1 -6103.53,E2 -6103.53} C_VEL
LIN {X 0,Y 495.787,Z 568.727,A -85,B 0,C 180,E1 -6106.055,E2 -6106.055} C_VEL
LIN {X 0,Y 495.865,Z 568.721,A -85,B 0,C 180,E1 -6108.555,E2 -6108.555} C_VEL
LIN {X 0,Y 495.864,Z 568.715,A -85,B 0,C 180,E1 -6111.852,E2 -6111.852} C_VEL
LIN {X 0,Y 495.904,Z 568.715,A -85,B 0,C 180,E1 -6114.307,E2 -6114.307} C_VEL
LIN {X 0,Y 495.984,Z 568.697,A -85,B 0,C 180,E1 -6117.564,E2 -6117.564} C_VEL
LIN {X 0,Y 495.987,Z 568.701,A -85,B 0,C 180,E1 -6120,E2 -6120} C_VEL
LIN {X 0,Y 495.984,Z 568.706,A -85,B 0,C 180,E1 -6122.436,E2 -6122.436} C_VEL
LIN {X 0,Y 495.907,Z 568.708,A -85,B 0,C 180,E1 -6125.693,E2 -6125.693} C_VEL
LIN {X 0,Y 495.864,Z 568.715,A -85,B 0,C 180,E1 -6128.148,E2 -6128.148} C_VEL
LIN {X 0,Y 495.859,Z 568.712,A -85,B 0,C 180,E1 -6131.445,E2 -6131.445} C_VEL
LIN {X 0,Y 495.784,Z 568.726,A -85,B 0,C 180,E1 -6134.783,E2 -6134.783} C_VEL
LIN {X 0,Y 495.778,Z 568.721,A -85,B 0,C 180,E1 -6137.319,E2 -6137.319} C_VEL
LIN {X 0,Y 495.769,Z 568.724,A -85,B 0,C 180,E1 -6139.891,E2 -6139.891} C_VEL
LIN {X 0,Y 495.756,Z 568.729,A -85,B 0,C 180,E1 -6142.863,E2 -6142.863} C_VEL
LIN {X 0,Y 495.792,Z 568.726,A -85,B 0,C 180,E1 -6146.068,E2 -6146.068} C_VEL
LIN {X 0,Y 495.773,Z 568.729,A -85,B 0,C 180,E1 -6148.815,E2 -6148.815} C_VEL
LIN {X 0,Y 495.752,Z 568.728,A -85,B 0,C 180,E1 -6151.727,E2 -6151.727} C_VEL
LIN {X 0,Y 495.77,Z 568.732,A -85,B 0,C 180,E1 -6154.696,E2 -6154.696} C_VEL
LIN {X 0,Y 495.727,Z 568.731,A -85,B 0,C 180,E1 -6157.562,E2 -6157.562} C_VEL
LIN {X 0,Y 495.788,Z 568.725,A -85,B 0,C 180,E1 -6160.053,E2 -6160.053} C_VEL
LIN {X 0,Y 495.76,Z 568.73,A -85,B 0,C 180,E1 -6162.88,E2 -6162.88} C_VEL
LIN {X 0,Y 495.73,Z 568.734,A -85,B 0,C 180,E1 -6166,E2 -6166} C_VEL
LIN {X 0,Y 495.769,Z 568.726,A -85,B 0,C 180,E1 -6169.302,E2 -6169.302} C_VEL
LIN {X 0,Y 495.755,Z 568.728,A -85,B 0,C 180,E1 -6171.41,E2 -6171.41} C_VEL
LIN {X 0,Y 495.749,Z 568.736,A -85,B 0,C 180,E1 -6174.463,E2 -6174.463} C_VEL
LIN {X 0,Y 495.767,Z 568.728,A -85,B 0,C 180,E1 -6177.407,E2 -6177.407} C_VEL
LIN {X 0,Y 495.765,Z 568.732,A -85,B 0,C 180,E1 -6180.254,E2 -6180.254} C_VEL
LIN {X 0,Y 495.83,Z 568.909,A -85,B 0,C 180,E1 -6182.628,E2 -6182.628} C_VEL
LIN {X 0,Y 498.217,Z 580.991,A -85,B 0,C 180,E1 -6184.53,E2 -6184.53} C_VEL
LIN {X 0,Y 497.943,Z 593.995,A -85,B 0,C 180,E1 -6186.414,E2 -6186.414} C_VEL
LIN {X 0,Y 497.223,Z 615.834,A -85,B 0,C 180,E1 -6189.524,E2 -6189.524} C_VEL
LIN {X 0,Y 496.662,Z 635.511,A -85,B 0,C 180,E1 -6192.288,E2 -6192.288} C_VEL
LIN {X 0,Y 496.406,Z 647.475,A -85,B 0,C 180,E1 -6193.958,E2 -6193.958} C_VEL
LIN {X 0,Y 498.478,Z 663.542,A -85,B 0,C 180,E1 -6194.268,E2 -6194.268} C_VEL
LIN {X 0,Y 497.901,Z 757.001,A -85,B 0,C 180,E1 -6195.647,E2 -6195.647} C_VEL
LIN {X 0,Y 497.553,Z 770.326,A -85,B 0,C 180,E1 -6196.002,E2 -6196.002} C_VEL
LIN {X 0,Y 497.286,Z 783.156,A -85,B 0,C 180,E1 -6196.515,E2 -6196.515} C_VEL
LIN {X 0,Y 496.942,Z 794.605,A -85,B 0,C 180,E1 -6197.132,E2 -6197.132} C_VEL
LIN {X 0,Y 496.557,Z 806.37,A -85,B 0,C 180,E1 -6197.95,E2 -6197.95} C_VEL
LIN {X 0,Y 496.167,Z 816.986,A -85,B 0,C 180,E1 -6198.873,E2 -6198.873} C_VEL
LIN {X 0,Y 495.853,Z 825.676,A -85,B 0,C 180,E1 -6199.795,E2 -6199.795} C_VEL
LIN {X 0,Y 495.588,Z 833.698,A -85,B 0,C 180,E1 -6200.82,E2 -6200.82} C_VEL
LIN {X 0,Y 495.358,Z 841.543,A -85,B 0,C 180,E1 -6202.049,E2 -6202.049} C_VEL
LIN {X 0,Y 495.164,Z 848.765,A -85,B 0,C 180,E1 -6203.48,E2 -6203.48} C_VEL
LIN {X 0,Y 495.126,Z 853.585,A -85,B 0,C 180,E1 -6204.706,E2 -6204.706} C_VEL
LIN {X 0,Y 495.131,Z 857.276,A -85,B 0,C 180,E1 -6205.93,E2 -6205.93} C_VEL
LIN {X 0,Y 495.046,Z 859.174,A -85,B 0,C 180,E1 -6206.745,E2 -6206.745} C_VEL
LIN {X 0,Y 495.053,Z 860.602,A -85,B 0,C 180,E1 -6207.559,E2 -6207.559} C_VEL
LIN {X 0,Y 494.927,Z 862.233,A -85,B 0,C 180,E1 -6209.186,E2 -6209.186} C_VEL
LIN {X 0,Y 494.92,Z 862.459,A -85,B 0,C 180,E1 -6210,E2 -6210} C_VEL
LIN {X 0,Y 494.926,Z 862.243,A -85,B 0,C 180,E1 -6210.814,E2 -6210.814} C_VEL
LIN {X 0,Y 495.053,Z 860.632,A -85,B 0,C 180,E1 -6212.441,E2 -6212.441} C_VEL
LIN {X 0,Y 495.046,Z 859.215,A -85,B 0,C 180,E1 -6213.255,E2 -6213.255} C_VEL
LIN {X 0,Y 495.052,Z 856.239,A -85,B 0,C 180,E1 -6214.478,E2 -6214.478} C_VEL
LIN {X 0,Y 495.167,Z 852.216,A -85,B 0,C 180,E1 -6215.702,E2 -6215.702} C_VEL
LIN {X 0,Y 495.249,Z 846.112,A -85,B 0,C 180,E1 -6217.112,E2 -6217.112} C_VEL
LIN {X 0,Y 495.451,Z 839.243,A -85,B 0,C 180,E1 -6218.36,E2 -6218.36} C_VEL
LIN {X 0,Y 495.667,Z 830.849,A -85,B 0,C 180,E1 -6219.59,E2 -6219.59} C_VEL
LIN {X 0,Y 495.986,Z 822.242,A -85,B 0,C 180,E1 -6220.615,E2 -6220.615} C_VEL
LIN {X 0,Y 496.391,Z 811.623,A -85,B 0,C 180,E1 -6221.639,E2 -6221.639} C_VEL
LIN {X 0,Y 496.705,Z 799.93,A -85,B 0,C 180,E1 -6222.546,E2 -6222.546} C_VEL
LIN {X 0,Y 497.103,Z 787.612,A -85,B 0,C 180,E1 -6223.281,E2 -6223.281} C_VEL
LIN {X 0,Y 497.525,Z 775.091,A -85,B 0,C 180,E1 -6223.842,E2 -6223.842} C_VEL
LIN {X 0,Y 497.815,Z 762.069,A -85,B 0,C 180,E1 -6224.251,E2 -6224.251} C_VEL
LIN {X 0,Y 498.034,Z 746.465,A -85,B 0,C 180,E1 -6224.532,E2 -6224.532} C_VEL
LIN {X 0,Y 498.401,Z 660.566,A -85,B 0,C 180,E1 -6225.787,E2 -6225.787} C_VEL
LIN {X 0,Y 496.717,Z 647.082,A -85,B 0,C 180,E1 -6226.051,E2 -6226.051} C_VEL
LIN {X 0,Y 497.482,Z 619.986,A -85,B 0,C 180,E1 -6229.389,E2 -6229.389} C_VEL
LIN {X 0,Y 498.248,Z 595.848,A -85,B 0,C 180,E1 -6232.386,E2 -6232.386} C_VEL
LIN {X 0,Y 498.666,Z 582.11,A -85,B 0,C 180,E1 -6234.123,E2 -6234.123} C_VEL
LIN {X 0,Y 495.855,Z 568.721,A -85,B 0,C 180,E1 -6236.007,E2 -6236.007} C_VEL
LIN {X 0,Y 495.772,Z 568.727,A -85,B 0,C 180,E1 -6238.814,E2 -6238.814} C_VEL
LIN {X 0,Y 495.755,Z 568.734,A -85,B 0,C 180,E1 -6241.725,E2 -6241.725} C_VEL
LIN {X 0,Y 495.776,Z 568.726,A -85,B 0,C 180,E1 -6244.695,E2 -6244.695} C_VEL
LIN {X 0,Y 495.729,Z 568.733,A -85,B 0,C 180,E1 -6247.561,E2 -6247.561} C_VEL
LIN {X 0,Y 495.777,Z 568.725,A -85,B 0,C 180,E1 -6250.698,E2 -6250.698} C_VEL
LIN {X 0,Y 495.73,Z 568.737,A -85,B 0,C 180,E1 -6254,E2 -6254} C_VEL
LIN {X 0,Y 495.759,Z 568.726,A -85,B 0,C 180,E1 -6257.12,E2 -6257.12} C_VEL
LIN {X 0,Y 495.786,Z 568.726,A -85,B 0,C 180,E1 -6260.365,E2 -6260.365} C_VEL
LIN {X 0,Y 495.728,Z 568.73,A -85,B 0,C 180,E1 -6263.456,E2 -6263.456} C_VEL
LIN {X 0,Y 495.754,Z 568.733,A -85,B 0,C 180,E1 -6266.435,E2 -6266.435} C_VEL
LIN {X 0,Y 495.75,Z 568.726,A -85,B 0,C 180,E1 -6269.312,E2 -6269.312} C_VEL
LIN {X 0,Y 495.775,Z 568.724,A -85,B 0,C 180,E1 -6272.108,E2 -6272.108} C_VEL
LIN {X 0,Y 495.781,Z 568.725,A -85,B 0,C 180,E1 -6274.832,E2 -6274.832} C_VEL
LIN {X 0,Y 495.74,Z 568.721,A -85,B 0,C 180,E1 -6277.494,E2 -6277.494} C_VEL
LIN {X 0,Y 495.769,Z 568.728,A -85,B 0,C 180,E1 -6280.109,E2 -6280.109} C_VEL
LIN {X 0,Y 495.778,Z 568.724,A -85,B 0,C 180,E1 -6282.681,E2 -6282.681} C_VEL
LIN {X 0,Y 495.78,Z 568.721,A -85,B 0,C 180,E1 -6285.217,E2 -6285.217} C_VEL
LIN {X 0,Y 495.845,Z 568.722,A -85,B 0,C 180,E1 -6288.555,E2 -6288.555} C_VEL
LIN {X 0,Y 495.864,Z 568.707,A -85,B 0,C 180,E1 -6291.852,E2 -6291.852} C_VEL
LIN {X 0,Y 495.908,Z 568.711,A -85,B 0,C 180,E1 -6294.307,E2 -6294.307} C_VEL
LIN {X 0,Y 495.984,Z 568.692,A -85,B 0,C 180,E1 -6297.564,E2 -6297.564} C_VEL
LIN {X 0,Y 495.987,Z 568.695,A -85,B 0,C 180,E1 -6300,E2 -6300} C_VEL
LIN {X 0,Y 495.984,Z 568.703,A -85,B 0,C 180,E1 -6302.436,E2 -6302.436} C_VEL
LIN {X 0,Y 495.897,Z 568.701,A -85,B 0,C 180,E1 -6305.693,E2 -6305.693} C_VEL
LIN {X 0,Y 495.864,Z 568.713,A -85,B 0,C 180,E1 -6308.148,E2 -6308.148} C_VEL
LIN {X 0,Y 495.845,Z 568.712,A -85,B 0,C 180,E1 -6311.445,E2 -6311.445} C_VEL
LIN {X 0,Y 495.78,Z 568.728,A -85,B 0,C 180,E1 -6314.783,E2 -6314.783} C_VEL
LIN {X 0,Y 495.778,Z 568.724,A -85,B 0,C 180,E1 -6317.319,E2 -6317.319} C_VEL
LIN {X 0,Y 495.769,Z 568.722,A -85,B 0,C 180,E1 -6319.891,E2 -6319.891} C_VEL
LIN {X 0,Y 495.752,Z 568.734,A -85,B 0,C 180,E1 -6322.862,E2 -6322.862} C_VEL
LIN {X 0,Y 495.791,Z 568.721,A -85,B 0,C 180,E1 -6326.068,E2 -6326.068} C_VEL
LIN {X 0,Y 495.773,Z 568.729,A -85,B 0,C 180,E1 -6328.815,E2 -6328.815} C_VEL
LIN {X 0,Y 495.752,Z 568.729,A -85,B 0,C 180,E1 -6331.727,E2 -6331.727} C_VEL
LIN {X 0,Y 495.769,Z 568.724,A -85,B 0,C 180,E1 -6334.696,E2 -6334.696} C_VEL
LIN {X 0,Y 495.727,Z 568.734,A -85,B 0,C 180,E1 -6337.562,E2 -6337.562} C_VEL
LIN {X 0,Y 495.761,Z 568.726,A -85,B 0,C 180,E1 -6340.701,E2 -6340.701} C_VEL
LIN {X 0,Y 495.73,Z 568.733,A -85,B 0,C 180,E1 -6343.696,E2 -6343.696} C_VEL
LIN {X 0,Y 495.724,Z 568.73,A -85,B 0,C 180,E1 -6346.306,E2 -6346.306} C_VEL
LIN {X 0,Y 495.763,Z 568.73,A -85,B 0,C 180,E1 -6349.301,E2 -6349.301} C_VEL
LIN {X 0,Y 495.729,Z 568.727,A -85,B 0,C 180,E1 -6352.439,E2 -6352.439} C_VEL
LIN {X 0,Y 495.783,Z 568.731,A -85,B 0,C 180,E1 -6355.458,E2 -6355.458} C_VEL
LIN {X 0,Y 495.755,Z 568.728,A -85,B 0,C 180,E1 -6358.365,E2 -6358.365} C_VEL
LIN {X 0,Y 495.753,Z 568.73,A -85,B 0,C 180,E1 -6360.773,E2 -6360.773} C_VEL
LIN {X 0,Y 495.627,Z 569.33,A -85,B 0,C 180,E1 -6361.077,E2 -6361.077} C_VEL
LIN {X 0,Y 495.191,Z 571.397,A -85,B 0,C 180,E1 -6361.423,E2 -6361.423} C_VEL
LIN {X 0,Y 494.414,Z 575.201,A -85,B 0,C 180,E1 -6361.756,E2 -6361.756} C_VEL
LIN {X 0,Y 493.361,Z 580.867,A -85,B 0,C 180,E1 -6362.014,E2 -6362.014} C_VEL
LIN {X 0,Y 492.338,Z 587.441,A -85,B 0,C 180,E1 -6362.18,E2 -6362.18} C_VEL
LIN {X 0,Y 491.734,Z 596.411,A -85,B 0,C 180,E1 -6362.326,E2 -6362.326} C_VEL
LIN {X 0,Y 491.196,Z 673.289,A -85,B 0,C 180,E1 -6363.47,E2 -6363.47} C_VEL
LIN {X 0,Y 490.965,Z 686.302,A -85,B 0,C 180,E1 -6363.814,E2 -6363.814} C_VEL
LIN {X 0,Y 490.765,Z 698.225,A -85,B 0,C 180,E1 -6364.291,E2 -6364.291} C_VEL
LIN {X 0,Y 490.456,Z 709.221,A -85,B 0,C 180,E1 -6364.881,E2 -6364.881} C_VEL
LIN {X 0,Y 490.06,Z 720.418,A -85,B 0,C 180,E1 -6365.651,E2 -6365.651} C_VEL
LIN {X 0,Y 489.617,Z 731.295,A -85,B 0,C 180,E1 -6366.591,E2 -6366.591} C_VEL
LIN {X 0,Y 489.248,Z 740.83,A -85,B 0,C 180,E1 -6367.625,E2 -6367.625} C_VEL
LIN {X 0,Y 488.925,Z 749.064,A -85,B 0,C 180,E1 -6368.719,E2 -6368.719} C_VEL
LIN {X 0,Y 488.573,Z 757.036,A -85,B 0,C 180,E1 -6370.024,E2 -6370.024} C_VEL
LIN {X 0,Y 488.417,Z 762.372,A -85,B 0,C 180,E1 -6371.11,E2 -6371.11} C_VEL
LIN {X 0,Y 488.228,Z 767.471,A -85,B 0,C 180,E1 -6372.405,E2 -6372.405} C_VEL
LIN {X 0,Y 488.118,Z 771.34,A -85,B 0,C 180,E1 -6373.695,E2 -6373.695} C_VEL
LIN {X 0,Y 488.019,Z 774.122,A -85,B 0,C 180,E1 -6374.977,E2 -6374.977} C_VEL
LIN {X 0,Y 487.956,Z 775.413,A -85,B 0,C 180,E1 -6375.827,E2 -6375.827} C_VEL
LIN {X 0,Y 487.921,Z 776.302,A -85,B 0,C 180,E1 -6376.676,E2 -6376.676} C_VEL
LIN {X 0,Y 487.943,Z 776.744,A -85,B 0,C 180,E1 -6377.523,E2 -6377.523} C_VEL
LIN {X 0,Y 487.974,Z 776.775,A -85,B 0,C 180,E1 -6378.368,E2 -6378.368} C_VEL
LIN {X 0,Y 488.004,Z 776.42,A -85,B 0,C 180,E1 -6379.21,E2 -6379.21} C_VEL
LIN {X 0,Y 487.934,Z 775.677,A -85,B 0,C 180,E1 -6380.047,E2 -6380.047} C_VEL
LIN {X 0,Y 488.055,Z 772.894,A -85,B 0,C 180,E1 -6381.721,E2 -6381.721} C_VEL
LIN {X 0,Y 488.201,Z 769.69,A -85,B 0,C 180,E1 -6382.972,E2 -6382.972} C_VEL
LIN {X 0,Y 488.263,Z 765.461,A -85,B 0,C 180,E1 -6384.217,E2 -6384.217} C_VEL
LIN {X 0,Y 488.463,Z 759.033,A -85,B 0,C 180,E1 -6385.668,E2 -6385.668} C_VEL
LIN {X 0,Y 488.711,Z 752.023,A -85,B 0,C 180,E1 -6386.909,E2 -6386.909} C_VEL
LIN {X 0,Y 489.089,Z 743.332,A -85,B 0,C 180,E1 -6388.147,E2 -6388.147} C_VEL
LIN {X 0,Y 489.519,Z 733.337,A -85,B 0,C 180,E1 -6389.28,E2 -6389.28} C_VEL
LIN {X 0,Y 489.854,Z 723.277,A -85,B 0,C 180,E1 -6390.206,E2 -6390.206} C_VEL
LIN {X 0,Y 490.298,Z 712.044,A -85,B 0,C 180,E1 -6391.027,E2 -6391.027} C_VEL
LIN {X 0,Y 490.739,Z 699.206,A -85,B 0,C 180,E1 -6391.744,E2 -6391.744} C_VEL
LIN {X 0,Y 491.019,Z 686.722,A -85,B 0,C 180,E1 -6392.256,E2 -6392.256} C_VEL
LIN {X 0,Y 491.214,Z 674.638,A -85,B 0,C 180,E1 -6392.588,E2 -6392.588} C_VEL
LIN {X 0,Y 491.501,Z 631.068,A -85,B 0,C 180,E1 -6393.253,E2 -6393.253} C_VEL
LIN {X 0,Y 491.736,Z 578.249,A -85,B 0,C 180,E1 -6394.034,E2 -6394.034} C_VEL
LIN {X 0,Y 488.712,Z 569.612,A -85,B 0,C 180,E1 -6394.278,E2 -6394.278} C_VEL
LIN {X 0,Y 488.821,Z 569.595,A -85,B 0,C 180,E1 -6396.605,E2 -6396.605} C_VEL
LIN {X 0,Y 488.778,Z 569.597,A -85,B 0,C 180,E1 -6399.1,E2 -6399.1} C_VEL
LIN {X 0,Y 488.821,Z 569.598,A -85,B 0,C 180,E1 -6402.131,E2 -6402.131} C_VEL
LIN {X 0,Y 488.779,Z 569.599,A -85,B 0,C 180,E1 -6405.555,E2 -6405.555} C_VEL
LIN {X 0,Y 488.757,Z 569.602,A -85,B 0,C 180,E1 -6408.442,E2 -6408.442} C_VEL
LIN {X 0,Y 488.708,Z 569.604,A -85,B 0,C 180,E1 -6411.07,E2 -6411.07} C_VEL
LIN {X 0,Y 488.677,Z 569.613,A -85,B 0,C 180,E1 -6413.746,E2 -6413.746} C_VEL
LIN {X 0,Y 488.792,Z 569.596,A -85,B 0,C 180,E1 -6416.943,E2 -6416.943} C_VEL
LIN {X 0,Y 488.773,Z 569.603,A -85,B 0,C 180,E1 -6419.799,E2 -6419.799} C_VEL
LIN {X 0,Y 491.843,Z 578.86,A -85,B 0,C 180,E1 -6420.071,E2 -6420.071} C_VEL
LIN {X 0,Y 491.101,Z 674.47,A -85,B 0,C 180,E1 -6421.519,E2 -6421.519} C_VEL
LIN {X 0,Y 490.899,Z 688.604,A -85,B 0,C 180,E1 -6421.925,E2 -6421.925} C_VEL
LIN {X 0,Y 490.62,Z 700.946,A -85,B 0,C 180,E1 -6422.457,E2 -6422.457} C_VEL
LIN {X 0,Y 490.277,Z 712.401,A -85,B 0,C 180,E1 -6423.119,E2 -6423.119} C_VEL
LIN {X 0,Y 489.889,Z 723.393,A -85,B 0,C 180,E1 -6423.926,E2 -6423.926} C_VEL
LIN {X 0,Y 489.545,Z 732.94,A -85,B 0,C 180,E1 -6424.795,E2 -6424.795} C_VEL
LIN {X 0,Y 489.144,Z 742.288,A -85,B 0,C 180,E1 -6425.837,E2 -6425.837} C_VEL
LIN {X 0,Y 488.848,Z 750.33,A -85,B 0,C 180,E1 -6426.941,E2 -6426.941} C_VEL
LIN {X 0,Y 488.53,Z 757.848,A -85,B 0,C 180,E1 -6428.213,E2 -6428.213} C_VEL
LIN {X 0,Y 488.348,Z 764.028,A -85,B 0,C 180,E1 -6429.529,E2 -6429.529} C_VEL
LIN {X 0,Y 488.17,Z 769.104,A -85,B 0,C 180,E1 -6430.922,E2 -6430.922} C_VEL
LIN {X 0,Y 488.03,Z 773.405,A -85,B 0,C 180,E1 -6432.596,E2 -6432.596} C_VEL
LIN {X 0,Y 487.947,Z 775.581,A -85,B 0,C 180,E1 -6433.932,E2 -6433.932} C_VEL
LIN {X 0,Y 487.893,Z 776.621,A -85,B 0,C 180,E1 -6435.103,E2 -6435.103} C_VEL
LIN {X 0,Y 487.877,Z 776.878,A -85,B 0,C 180,E1 -6436.255,E2 -6436.255} C_VEL
LIN {X 0,Y 487.942,Z 776.398,A -85,B 0,C 180,E1 -6437.393,E2 -6437.393} C_VEL
LIN {X 0,Y 487.954,Z 775.183,A -85,B 0,C 180,E1 -6438.506,E2 -6438.506} C_VEL
LIN {X 0,Y 488.026,Z 772.959,A -85,B 0,C 180,E1 -6439.749,E2 -6439.749} C_VEL
LIN {X 0,Y 488.158,Z 769.667,A -85,B 0,C 180,E1 -6441.025,E2 -6441.025} C_VEL
LIN {X 0,Y 488.361,Z 764.143,A -85,B 0,C 180,E1 -6442.574,E2 -6442.574} C_VEL
LIN {X 0,Y 488.53,Z 758.173,A -85,B 0,C 180,E1 -6443.855,E2 -6443.855} C_VEL
LIN {X 0,Y 488.792,Z 751.289,A -85,B 0,C 180,E1 -6445.039,E2 -6445.039} C_VEL
LIN {X 0,Y 489.186,Z 742.877,A -85,B 0,C 180,E1 -6446.212,E2 -6446.212} C_VEL
LIN {X 0,Y 489.526,Z 733.178,A -85,B 0,C 180,E1 -6447.303,E2 -6447.303} C_VEL
LIN {X 0,Y 489.941,Z 723.45,A -85,B 0,C 180,E1 -6448.186,E2 -6448.186} C_VEL
LIN {X 0,Y 490.26,Z 713.381,A -85,B 0,C 180,E1 -6448.931,E2 -6448.931} C_VEL
